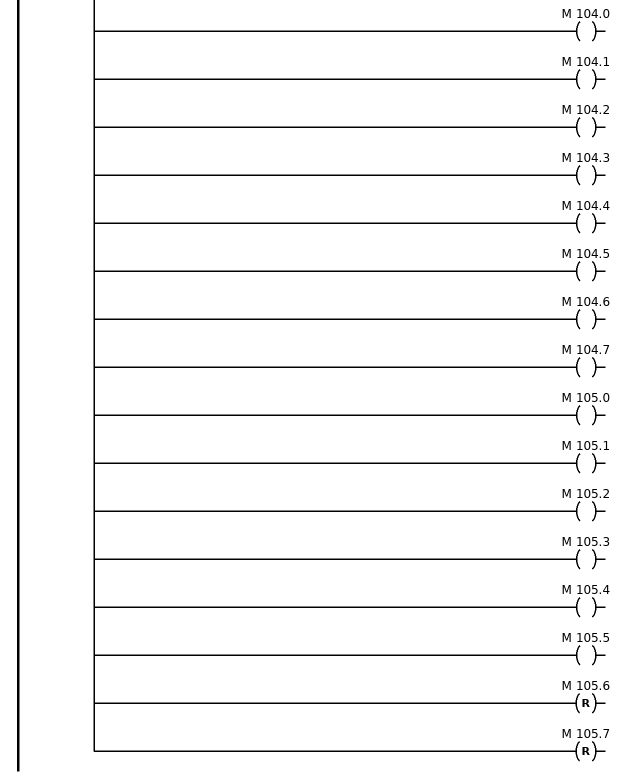
[picture p239: FC51 - TYPE TOOL networks 18-18]
NETWORK
TITLE = Error visible
      A     M 90.2;
      JCN   v10;
      SET;
      =     M 104.0;
      =     M 104.1;
      =     M 104.2;
      =     M 104.3;
      =     M 104.4;
      =     M 104.5;
      =     M 104.6;
      =     M 104.7;
      =     M 105.0;
      R     M 105.1;
      R     M 105.2;
      R     M 105.3;
      R     M 105.4;
      R     M 105.5;
      =     M 105.6;
      R     M 105.7;
      JU    next;
v10:  NOP   0;
      A     M 90.0;
      JCN   v11;
      SET;
      =     M 104.0;
      =     M 104.1;
      =     M 104.2;
      =     M 104.3;
      =     M 104.4;
      =     M 104.5;
      =     M 104.6;
      =     M 104.7;
      =     M 105.0;
      =     M 105.1;
      R     M 105.2;
      R     M 105.3;
      R     M 105.4;
      =     M 105.5;
      R     M 105.6;
      R     M 105.7;
      JU    next;
v11:  NOP   0;
      A     M 90.1;
      JCN   v13;
      SET;
      =     M 104.0;
      =     M 104.1;
      =     M 104.2;
      =     M 104.3;
      =     M 104.4;
      =     M 104.5;
      =     M 104.6;
      =     M 104.7;
      =     M 105.0;
      =     M 105.1;
      =     M 105.2;
      R     M 105.3;
      R     M 105.4;
      =     M 105.5;
      R     M 105.6;
      R     M 105.7;
      JU    next;
v13:  NOP   0;
      A     M 90.3;
      JCN   next;
      =     M 104.0;
      =     M 104.1;
      =     M 104.2;
      =     M 104.3;
      =     M 104.4;
      =     M 104.5;
      =     M 104.6;
      =     M 104.7;
      =     M 105.0;
      =     M 105.1;
      =     M 105.2;
      =     M 105.3;
      =     M 105.4;
      =     M 105.5;
      R     M 105.6;
      R     M 105.7;
next: NOP   0;
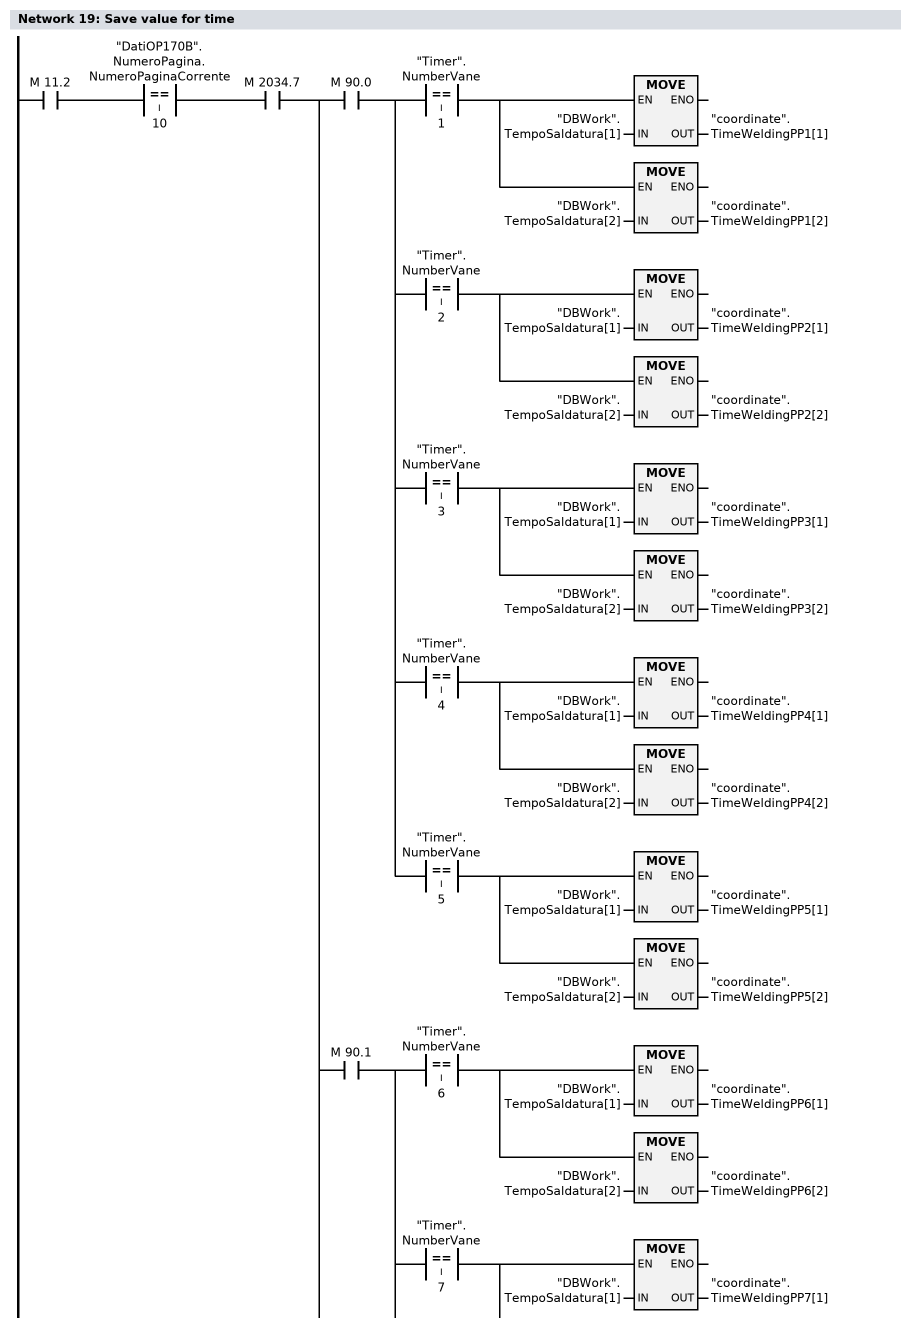
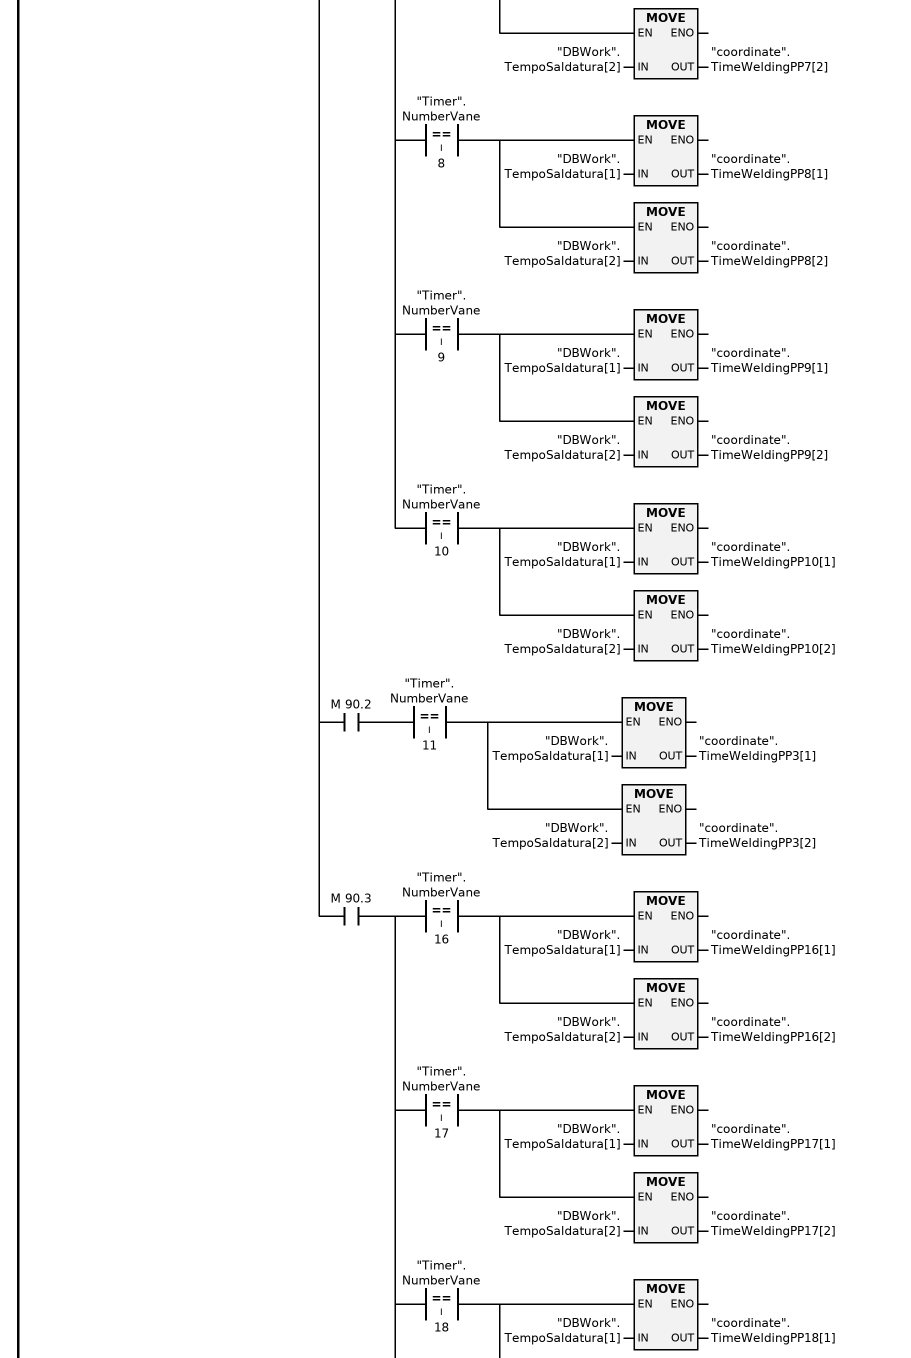
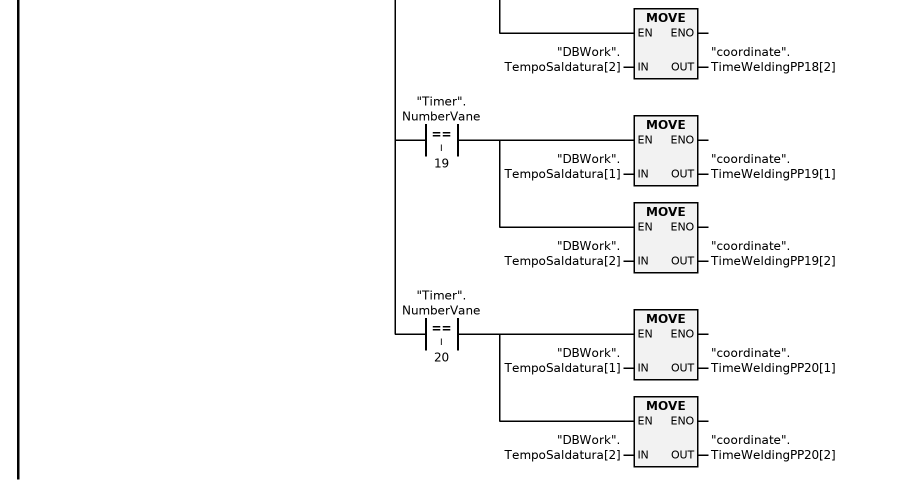
NETWORK
TITLE = Save value for time
      A     M 11.2;
      A(;
      L     "DatiOP170B".NumeroPagina.NumeroPaginaCorrente;
      L     10;
      ==I;
      );
      A     M 2034.7;
      =     L 0.0;
      A     L 0.0;
      A     M 90.0;
      =     L 0.1;
      A     L 0.1;
      A(;
      L     "Timer".NumberVane;
      L     1;
      ==I;
      );
      =     L 0.2;
      A     L 0.2;
      JNB   _0c6;
      L     "DBWork".TempoSaldatura[1];
      T     "coordinate".TimeWeldingPP1[1];
_0c6: NOP   0;
      A     L 0.2;
      JNB   _0c7;
      L     "DBWork".TempoSaldatura[2];
      T     "coordinate".TimeWeldingPP1[2];
_0c7: NOP   0;
      A     L 0.1;
      A(;
      L     "Timer".NumberVane;
      L     2;
      ==I;
      );
      =     L 0.2;
      A     L 0.2;
      JNB   _0c8;
      L     "DBWork".TempoSaldatura[1];
      T     "coordinate".TimeWeldingPP2[1];
_0c8: NOP   0;
      A     L 0.2;
      JNB   _0c9;
      L     "DBWork".TempoSaldatura[2];
      T     "coordinate".TimeWeldingPP2[2];
_0c9: NOP   0;
      A     L 0.1;
      A(;
      L     "Timer".NumberVane;
      L     3;
      ==I;
      );
      =     L 0.2;
      A     L 0.2;
      JNB   _0ca;
      L     "DBWork".TempoSaldatura[1];
      T     "coordinate".TimeWeldingPP3[1];
_0ca: NOP   0;
      A     L 0.2;
      JNB   _0cb;
      L     "DBWork".TempoSaldatura[2];
      T     "coordinate".TimeWeldingPP3[2];
_0cb: NOP   0;
      A     L 0.1;
      A(;
      L     "Timer".NumberVane;
      L     4;
      ==I;
      );
      =     L 0.2;
      A     L 0.2;
      JNB   _0cc;
      L     "DBWork".TempoSaldatura[1];
      T     "coordinate".TimeWeldingPP4[1];
_0cc: NOP   0;
      A     L 0.2;
      JNB   _0cd;
      L     "DBWork".TempoSaldatura[2];
      T     "coordinate".TimeWeldingPP4[2];
_0cd: NOP   0;
      A     L 0.1;
      A(;
      L     "Timer".NumberVane;
      L     5;
      ==I;
      );
      =     L 0.2;
      A     L 0.2;
      JNB   _0ce;
      L     "DBWork".TempoSaldatura[1];
      T     "coordinate".TimeWeldingPP5[1];
_0ce: NOP   0;
      A     L 0.2;
      JNB   _0cf;
      L     "DBWork".TempoSaldatura[2];
      T     "coordinate".TimeWeldingPP5[2];
_0cf: NOP   0;
      A     L 0.0;
      A     M 90.1;
      =     L 0.1;
      A     L 0.1;
      A(;
      L     "Timer".NumberVane;
      L     6;
      ==I;
      );
      =     L 0.2;
      A     L 0.2;
      JNB   _0d0;
      L     "DBWork".TempoSaldatura[1];
      T     "coordinate".TimeWeldingPP6[1];
_0d0: NOP   0;
      A     L 0.2;
      JNB   _0d1;
      L     "DBWork".TempoSaldatura[2];
      T     "coordinate".TimeWeldingPP6[2];
_0d1: NOP   0;
      A     L 0.1;
      A(;
      L     "Timer".NumberVane;
      L     7;
      ==I;
      );
      =     L 0.2;
      A     L 0.2;
      JNB   _0d2;
      L     "DBWork".TempoSaldatura[1];
      T     "coordinate".TimeWeldingPP7[1];
_0d2: NOP   0;
      A     L 0.2;
      JNB   _0d3;
      L     "DBWork".TempoSaldatura[2];
      T     "coordinate".TimeWeldingPP7[2];
_0d3: NOP   0;
      A     L 0.1;
      A(;
      L     "Timer".NumberVane;
      L     8;
      ==I;
      );
      =     L 0.2;
      A     L 0.2;
      JNB   _0d4;
      L     "DBWork".TempoSaldatura[1];
      T     "coordinate".TimeWeldingPP8[1];
_0d4: NOP   0;
      A     L 0.2;
      JNB   _0d5;
      L     "DBWork".TempoSaldatura[2];
      T     "coordinate".TimeWeldingPP8[2];
_0d5: NOP   0;
      A     L 0.1;
      A(;
      L     "Timer".NumberVane;
      L     9;
      ==I;
      );
      =     L 0.2;
      A     L 0.2;
      JNB   _0d6;
      L     "DBWork".TempoSaldatura[1];
      T     "coordinate".TimeWeldingPP9[1];
_0d6: NOP   0;
      A     L 0.2;
      JNB   _0d7;
      L     "DBWork".TempoSaldatura[2];
      T     "coordinate".TimeWeldingPP9[2];
_0d7: NOP   0;
      A     L 0.1;
      A(;
      L     "Timer".NumberVane;
      L     10;
      ==I;
      );
      =     L 0.2;
      A     L 0.2;
      JNB   _0d8;
      L     "DBWork".TempoSaldatura[1];
      T     "coordinate".TimeWeldingPP10[1];
_0d8: NOP   0;
      A     L 0.2;
      JNB   _0d9;
      L     "DBWork".TempoSaldatura[2];
      T     "coordinate".TimeWeldingPP10[2];
_0d9: NOP   0;
      A     L 0.0;
      A     M 90.2;
      A(;
      L     "Timer".NumberVane;
      L     11;
      ==I;
      );
      =     L 0.1;
      A     L 0.1;
      JNB   _0da;
      L     "DBWork".TempoSaldatura[1];
      T     "coordinate".TimeWeldingPP3[1];
_0da: NOP   0;
      A     L 0.1;
      JNB   _0db;
      L     "DBWork".TempoSaldatura[2];
      T     "coordinate".TimeWeldingPP3[2];
_0db: NOP   0;
      A     L 0.0;
      A     M 90.3;
      =     L 0.1;
      A     L 0.1;
      A(;
      L     "Timer".NumberVane;
      L     16;
      ==I;
      );
      =     L 0.2;
      A     L 0.2;
      JNB   _0dc;
      L     "DBWork".TempoSaldatura[1];
      T     "coordinate".TimeWeldingPP16[1];
_0dc: NOP   0;
      A     L 0.2;
      JNB   _0dd;
      L     "DBWork".TempoSaldatura[2];
      T     "coordinate".TimeWeldingPP16[2];
_0dd: NOP   0;
      A     L 0.1;
      A(;
      L     "Timer".NumberVane;
      L     17;
      ==I;
      );
      =     L 0.2;
      A     L 0.2;
      JNB   _0de;
      L     "DBWork".TempoSaldatura[1];
      T     "coordinate".TimeWeldingPP17[1];
_0de: NOP   0;
      A     L 0.2;
      JNB   _0df;
      L     "DBWork".TempoSaldatura[2];
      T     "coordinate".TimeWeldingPP17[2];
_0df: NOP   0;
      A     L 0.1;
      A(;
      L     "Timer".NumberVane;
      L     18;
      ==I;
      );
      =     L 0.2;
      A     L 0.2;
      JNB   _0e0;
      L     "DBWork".TempoSaldatura[1];
      T     "coordinate".TimeWeldingPP18[1];
_0e0: NOP   0;
      A     L 0.2;
      JNB   _0e1;
      L     "DBWork".TempoSaldatura[2];
      T     "coordinate".TimeWeldingPP18[2];
_0e1: NOP   0;
      A     L 0.1;
      A(;
      L     "Timer".NumberVane;
      L     19;
      ==I;
      );
      =     L 0.2;
      A     L 0.2;
      JNB   _0e2;
      L     "DBWork".TempoSaldatura[1];
      T     "coordinate".TimeWeldingPP19[1];
_0e2: NOP   0;
      A     L 0.2;
      JNB   _0e3;
      L     "DBWork".TempoSaldatura[2];
      T     "coordinate".TimeWeldingPP19[2];
_0e3: NOP   0;
      A     L 0.1;
      A(;
      L     "Timer".NumberVane;
      L     20;
      ==I;
      );
      =     L 0.2;
      A     L 0.2;
      JNB   _0e4;
      L     "DBWork".TempoSaldatura[1];
      T     "coordinate".TimeWeldingPP20[1];
_0e4: NOP   0;
      A     L 0.2;
      JNB   _0e5;
      L     "DBWork".TempoSaldatura[2];
      T     "coordinate".TimeWeldingPP20[2];
_0e5: NOP   0;
NETWORK
TITLE =
NETWORK
TITLE = load value for selected point, use it in auto, teach in and weld
//carico le coordinate del punto selezionato per fare le saldature in automatico 
//per il teachIn e per il test di salsatura
      A     M 1.1;
      =     L 0.0;
      A     L 0.0;
      A(;
      A(;
      L     "DBWork".PP[1].NumSaldaturaAtt;
      L     0;
      ==I;
      );
      A     M 11.4;
      O;
      A     M 11.2;
      A(;
      L     "DatiOP170B".PointWeldingTeachIn;
      L     1;
      ==I;
      );
      A(;
      O(;
      L     "DatiOP170B".NumeroPagina.NumeroPaginaCorrente;
      L     5;
      ==I;
      );
      O(;
      L     "DatiOP170B".NumeroPagina.NumeroPaginaCorrente;
      L     11;
      ==I;
      );
      );
      );
      =     L 0.1;
      A(;
      A     L 0.1;
      A     "DBWork".RotationTable;
      JNB   _0e6;
      L     "DBWork".CoordSaldatura[1].X1;
      T     MD 588;
      SET;
      SAVE;
      CLR;
_0e6: A     BR;
      );
      JNB   _0e7;
      L     "DBWork".CoordSaldatura[1].Y1;
      T     MD 592;
_0e7: NOP   0;
      A(;
      A     L 0.1;
      AN    "DBWork".RotationTable;
      JNB   _0e8;
      L     "DBWork".CoordSaldatura[1].X2;
      T     MD 588;
      SET;
      SAVE;
      CLR;
_0e8: A     BR;
      );
      JNB   _0e9;
      L     "DBWork".CoordSaldatura[1].Y2;
      T     MD 592;
_0e9: NOP   0;
      A     L 0.0;
      A(;
      A(;
      L     "DBWork".PP[1].NumSaldaturaAtt;
      L     1;
      ==I;
      );
      A     M 11.4;
      O;
      A     M 11.2;
      A(;
      L     "DatiOP170B".PointWeldingTeachIn;
      L     2;
      ==I;
      );
      A(;
      O(;
      L     "DatiOP170B".NumeroPagina.NumeroPaginaCorrente;
      L     5;
      ==I;
      );
      O(;
      L     "DatiOP170B".NumeroPagina.NumeroPaginaCorrente;
      L     11;
      ==I;
      );
      );
      );
      =     L 0.1;
      A(;
      A     L 0.1;
      A     "DBWork".RotationTable;
      JNB   _0ea;
      L     "DBWork".CoordSaldatura[2].X1;
      T     MD 588;
      SET;
      SAVE;
      CLR;
_0ea: A     BR;
      );
      JNB   _0eb;
      L     "DBWork".CoordSaldatura[2].Y1;
      T     MD 592;
_0eb: NOP   0;
      A(;
      A     L 0.1;
      AN    "DBWork".RotationTable;
      JNB   _0ec;
      L     "DBWork".CoordSaldatura[2].X2;
      T     MD 588;
      SET;
      SAVE;
      CLR;
_0ec: A     BR;
      );
      JNB   _0ed;
      L     "DBWork".CoordSaldatura[2].Y2;
      T     MD 592;
_0ed: NOP   0;
      A     L 0.0;
      A(;
      A(;
      L     "DBWork".PP[1].NumSaldaturaAtt;
      L     2;
      ==I;
      );
      A     M 11.4;
      O;
      A     M 11.2;
      A(;
      L     "DatiOP170B".PointWeldingTeachIn;
      L     3;
      ==I;
      );
      A(;
      O(;
      L     "DatiOP170B".NumeroPagina.NumeroPaginaCorrente;
      L     5;
      ==I;
      );
      O(;
      L     "DatiOP170B".NumeroPagina.NumeroPaginaCorrente;
      L     11;
      ==I;
      );
      );
      );
      =     L 0.1;
      A(;
      A     L 0.1;
      A     "DBWork".RotationTable;
      JNB   _0ee;
      L     "DBWork".CoordSaldatura[3].X1;
      T     MD 588;
      SET;
      SAVE;
      CLR;
_0ee: A     BR;
      );
      JNB   _0ef;
      L     "DBWork".CoordSaldatura[3].Y1;
      T     MD 592;
_0ef: NOP   0;
      A(;
      A     L 0.1;
      AN    "DBWork".RotationTable;
      JNB   _0f0;
      L     "DBWork".CoordSaldatura[3].X2;
      T     MD 588;
      SET;
      SAVE;
      CLR;
_0f0: A     BR;
      );
      JNB   _0f1;
      L     "DBWork".CoordSaldatura[3].Y2;
      T     MD 592;
_0f1: NOP   0;
      A     L 0.0;
      A(;
      A(;
      L     "DBWork".PP[1].NumSaldaturaAtt;
      L     3;
      ==I;
      );
      A     M 11.4;
      O;
      A     M 11.2;
      A(;
      L     "DatiOP170B".PointWeldingTeachIn;
      L     4;
      ==I;
      );
      A(;
      O(;
      L     "DatiOP170B".NumeroPagina.NumeroPaginaCorrente;
      L     5;
      ==I;
      );
      O(;
      L     "DatiOP170B".NumeroPagina.NumeroPaginaCorrente;
      L     11;
      ==I;
      );
      );
      );
      =     L 0.1;
      A(;
      A     L 0.1;
      A     "DBWork".RotationTable;
      JNB   _0f2;
      L     "DBWork".CoordSaldatura[4].X1;
      T     MD 588;
      SET;
      SAVE;
      CLR;
_0f2: A     BR;
      );
      JNB   _0f3;
      L     "DBWork".CoordSaldatura[4].Y1;
      T     MD 592;
_0f3: NOP   0;
      A(;
      A     L 0.1;
      AN    "DBWork".RotationTable;
      JNB   _0f4;
      L     "DBWork".CoordSaldatura[4].X2;
      T     MD 588;
      SET;
      SAVE;
      CLR;
_0f4: A     BR;
      );
      JNB   _0f5;
      L     "DBWork".CoordSaldatura[4].Y2;
      T     MD 592;
_0f5: NOP   0;
      A     L 0.0;
      A(;
      A(;
      L     "DBWork".PP[1].NumSaldaturaAtt;
      L     4;
      ==I;
      );
      A     M 11.4;
      O;
      A     M 11.2;
      A(;
      L     "DatiOP170B".PointWeldingTeachIn;
      L     5;
      ==I;
      );
      A(;
      O(;
      L     "DatiOP170B".NumeroPagina.NumeroPaginaCorrente;
      L     5;
      ==I;
      );
      O(;
      L     "DatiOP170B".NumeroPagina.NumeroPaginaCorrente;
      L     11;
      ==I;
      );
      );
      );
      =     L 0.1;
      A(;
      A     L 0.1;
      A     "DBWork".RotationTable;
      JNB   _0f6;
      L     "DBWork".CoordSaldatura[5].X1;
      T     MD 588;
      SET;
      SAVE;
      CLR;
_0f6: A     BR;
      );
      JNB   _0f7;
      L     "DBWork".CoordSaldatura[5].Y1;
      T     MD 592;
_0f7: NOP   0;
      A(;
      A     L 0.1;
      AN    "DBWork".RotationTable;
      JNB   _0f8;
      L     "DBWork".CoordSaldatura[5].X2;
      T     MD 588;
      SET;
      SAVE;
      CLR;
_0f8: A     BR;
      );
      JNB   _0f9;
      L     "DBWork".CoordSaldatura[5].Y2;
      T     MD 592;
_0f9: NOP   0;
      A     L 0.0;
      A(;
      A(;
      L     "DBWork".PP[1].NumSaldaturaAtt;
      L     5;
      ==I;
      );
      A     M 11.4;
      O;
      A     M 11.2;
      A(;
      L     "DatiOP170B".PointWeldingTeachIn;
      L     6;
      ==I;
      );
      A(;
      O(;
      L     "DatiOP170B".NumeroPagina.NumeroPaginaCorrente;
      L     5;
      ==I;
      );
      O(;
      L     "DatiOP170B".NumeroPagina.NumeroPaginaCorrente;
      L     11;
      ==I;
      );
      );
      );
      =     L 0.1;
      A(;
      A     L 0.1;
      A     "DBWork".RotationTable;
      JNB   _0fa;
      L     "DBWork".CoordSaldatura[6].X1;
      T     MD 588;
      SET;
      SAVE;
      CLR;
_0fa: A     BR;
      );
      JNB   _0fb;
      L     "DBWork".CoordSaldatura[6].Y1;
      T     MD 592;
_0fb: NOP   0;
      A(;
      A     L 0.1;
      AN    "DBWork".RotationTable;
      JNB   _0fc;
      L     "DBWork".CoordSaldatura[6].X2;
      T     MD 588;
      SET;
      SAVE;
      CLR;
_0fc: A     BR;
      );
      JNB   _0fd;
      L     "DBWork".CoordSaldatura[6].Y2;
      T     MD 592;
_0fd: NOP   0;
      A     L 0.0;
      A(;
      A(;
      L     "DBWork".PP[1].NumSaldaturaAtt;
      L     6;
      ==I;
      );
      A     M 11.4;
      O;
      A     M 11.2;
      A(;
      L     "DatiOP170B".PointWeldingTeachIn;
      L     7;
      ==I;
      );
      A(;
      O(;
      L     "DatiOP170B".NumeroPagina.NumeroPaginaCorrente;
      L     5;
      ==I;
      );
      O(;
      L     "DatiOP170B".NumeroPagina.NumeroPaginaCorrente;
      L     11;
      ==I;
      );
      );
      );
      =     L 0.1;
      A(;
      A     L 0.1;
      A     "DBWork".RotationTable;
      JNB   _0fe;
      L     "DBWork".CoordSaldatura[7].X1;
      T     MD 588;
      SET;
      SAVE;
      CLR;
_0fe: A     BR;
      );
      JNB   _0ff;
      L     "DBWork".CoordSaldatura[7].Y1;
      T     MD 592;
_0ff: NOP   0;
      A(;
      A     L 0.1;
      AN    "DBWork".RotationTable;
      JNB   _100;
      L     "DBWork".CoordSaldatura[7].X2;
      T     MD 588;
      SET;
      SAVE;
      CLR;
_100: A     BR;
      );
      JNB   _101;
      L     "DBWork".CoordSaldatura[7].Y2;
      T     MD 592;
_101: NOP   0;
      A     L 0.0;
      A(;
      A(;
      L     "DBWork".PP[1].NumSaldaturaAtt;
      L     7;
      ==I;
      );
      A     M 11.4;
      O;
      A     M 11.2;
      A(;
      L     "DatiOP170B".PointWeldingTeachIn;
      L     8;
      ==I;
      );
      A(;
      O(;
      L     "DatiOP170B".NumeroPagina.NumeroPaginaCorrente;
      L     5;
      ==I;
      );
      O(;
      L     "DatiOP170B".NumeroPagina.NumeroPaginaCorrente;
      L     11;
      ==I;
      );
      );
      );
      =     L 0.1;
      A(;
      A     L 0.1;
      A     "DBWork".RotationTable;
      JNB   _102;
      L     "DBWork".CoordSaldatura[8].X1;
      T     MD 588;
      SET;
      SAVE;
      CLR;
_102: A     BR;
      );
      JNB   _103;
      L     "DBWork".CoordSaldatura[8].Y1;
      T     MD 592;
_103: NOP   0;
      A(;
      A     L 0.1;
      AN    "DBWork".RotationTable;
      JNB   _104;
      L     "DBWork".CoordSaldatura[8].X2;
      T     MD 588;
      SET;
      SAVE;
      CLR;
_104: A     BR;
      );
      JNB   _105;
      L     "DBWork".CoordSaldatura[8].Y2;
      T     MD 592;
_105: NOP   0;
      A     L 0.0;
      A(;
      A(;
      L     "DBWork".PP[1].NumSaldaturaAtt;
      L     8;
      ==I;
      );
      A     M 11.4;
      O;
      A     M 11.2;
      A(;
      L     "DatiOP170B".PointWeldingTeachIn;
      L     9;
      ==I;
      );
      A(;
      O(;
      L     "DatiOP170B".NumeroPagina.NumeroPaginaCorrente;
      L     5;
      ==I;
      );
      O(;
      L     "DatiOP170B".NumeroPagina.NumeroPaginaCorrente;
      L     11;
      ==I;
      );
      );
      );
      =     L 0.1;
      A(;
      A     L 0.1;
      A     "DBWork".RotationTable;
      JNB   _106;
      L     "DBWork".CoordSaldatura[9].X1;
      T     MD 588;
      SET;
      SAVE;
      CLR;
_106: A     BR;
      );
      JNB   _107;
      L     "DBWork".CoordSaldatura[9].Y1;
      T     MD 592;
_107: NOP   0;
      A(;
      A     L 0.1;
      AN    "DBWork".RotationTable;
      JNB   _108;
      L     "DBWork".CoordSaldatura[9].X2;
      T     MD 588;
      SET;
      SAVE;
      CLR;
_108: A     BR;
      );
      JNB   _109;
      L     "DBWork".CoordSaldatura[9].Y2;
      T     MD 592;
_109: NOP   0;
      A     L 0.0;
      A(;
      A(;
      L     "DBWork".PP[1].NumSaldaturaAtt;
      L     9;
      ==I;
      );
      A     M 11.4;
      O;
      A     M 11.2;
      A(;
      L     "DatiOP170B".PointWeldingTeachIn;
      L     10;
      ==I;
      );
      A(;
      O(;
      L     "DatiOP170B".NumeroPagina.NumeroPaginaCorrente;
      L     5;
      ==I;
      );
      O(;
      L     "DatiOP170B".NumeroPagina.NumeroPaginaCorrente;
      L     11;
      ==I;
      );
      );
      );
      =     L 0.1;
      A(;
      A     L 0.1;
      A     "DBWork".RotationTable;
      JNB   _10a;
      L     "DBWork".CoordSaldatura[10].X1;
      T     MD 588;
      SET;
      SAVE;
      CLR;
_10a: A     BR;
      );
      JNB   _10b;
      L     "DBWork".CoordSaldatura[10].Y1;
      T     MD 592;
_10b: NOP   0;
      A(;
      A     L 0.1;
      AN    "DBWork".RotationTable;
      JNB   _10c;
      L     "DBWork".CoordSaldatura[10].X2;
      T     MD 588;
      SET;
      SAVE;
      CLR;
_10c: A     BR;
      );
      JNB   _10d;
      L     "DBWork".CoordSaldatura[10].Y2;
      T     MD 592;
_10d: NOP   0;
      A     L 0.0;
      A(;
      A(;
      L     "DBWork".PP[1].NumSaldaturaAtt;
      L     10;
      ==I;
      );
      A     M 11.4;
      O;
      A     M 11.2;
      A(;
      L     "DatiOP170B".PointWeldingTeachIn;
      L     11;
      ==I;
      );
      A(;
      O(;
      L     "DatiOP170B".NumeroPagina.NumeroPaginaCorrente;
      L     5;
      ==I;
      );
      O(;
      L     "DatiOP170B".NumeroPagina.NumeroPaginaCorrente;
      L     11;
      ==I;
      );
      );
      );
      =     L 0.1;
      A(;
      A     L 0.1;
      A     "DBWork".RotationTable;
      JNB   _10e;
      L     "DBWork".CoordSaldatura[11].X1;
      T     MD 588;
      SET;
      SAVE;
      CLR;
_10e: A     BR;
      );
      JNB   _10f;
      L     "DBWork".CoordSaldatura[11].Y1;
      T     MD 592;
_10f: NOP   0;
      A(;
      A     L 0.1;
      AN    "DBWork".RotationTable;
      JNB   _110;
      L     "DBWork".CoordSaldatura[11].X2;
      T     MD 588;
      SET;
      SAVE;
      CLR;
_110: A     BR;
      );
      JNB   _111;
      L     "DBWork".CoordSaldatura[11].Y2;
      T     MD 592;
_111: NOP   0;
      A     L 0.0;
      A(;
      A(;
      L     "DBWork".PP[1].NumSaldaturaAtt;
      L     11;
      ==I;
      );
      A     M 11.4;
      O;
      A     M 11.2;
      A(;
      L     "DatiOP170B".PointWeldingTeachIn;
      L     12;
      ==I;
      );
      A(;
      O(;
      L     "DatiOP170B".NumeroPagina.NumeroPaginaCorrente;
      L     5;
      ==I;
      );
      O(;
      L     "DatiOP170B".NumeroPagina.NumeroPaginaCorrente;
      L     11;
      ==I;
      );
      );
      );
      =     L 0.1;
      A(;
      A     L 0.1;
      A     "DBWork".RotationTable;
      JNB   _112;
      L     "DBWork".CoordSaldatura[12].X1;
      T     MD 588;
      SET;
      SAVE;
      CLR;
_112: A     BR;
      );
      JNB   _113;
      L     "DBWork".CoordSaldatura[12].Y1;
      T     MD 592;
_113: NOP   0;
      A(;
      A     L 0.1;
      AN    "DBWork".RotationTable;
      JNB   _114;
      L     "DBWork".CoordSaldatura[12].X2;
      T     MD 588;
      SET;
      SAVE;
      CLR;
_114: A     BR;
      );
      JNB   _115;
      L     "DBWork".CoordSaldatura[12].Y2;
      T     MD 592;
_115: NOP   0;
      A     L 0.0;
      A(;
      A(;
      L     "DBWork".PP[1].NumSaldaturaAtt;
      L     12;
      ==I;
      );
      A     M 11.4;
      O;
      A     M 11.2;
      A(;
      L     "DatiOP170B".PointWeldingTeachIn;
      L     13;
      ==I;
      );
      A(;
      O(;
      L     "DatiOP170B".NumeroPagina.NumeroPaginaCorrente;
      L     5;
      ==I;
      );
      O(;
      L     "DatiOP170B".NumeroPagina.NumeroPaginaCorrente;
      L     11;
      ==I;
      );
      );
      );
      =     L 0.1;
      A(;
      A     L 0.1;
      A     "DBWork".RotationTable;
      JNB   _116;
      L     "DBWork".CoordSaldatura[13].X1;
      T     MD 588;
      SET;
      SAVE;
      CLR;
_116: A     BR;
      );
      JNB   _117;
      L     "DBWork".CoordSaldatura[13].Y1;
      T     MD 592;
_117: NOP   0;
      A(;
      A     L 0.1;
      AN    "DBWork".RotationTable;
      JNB   _118;
      L     "DBWork".CoordSaldatura[13].X2;
      T     MD 588;
      SET;
      SAVE;
      CLR;
_118: A     BR;
      );
      JNB   _119;
      L     "DBWork".CoordSaldatura[13].Y2;
      T     MD 592;
_119: NOP   0;
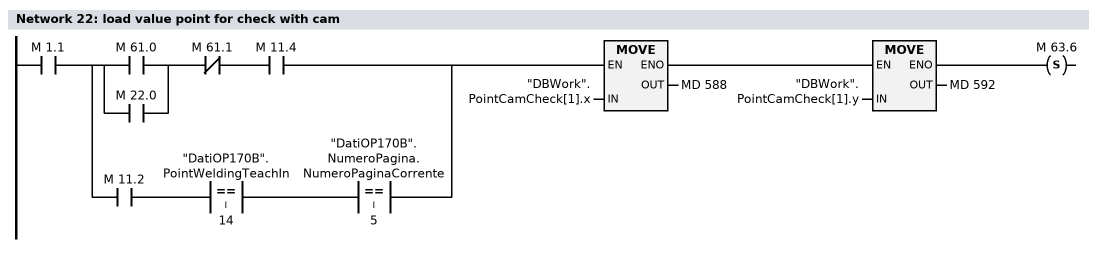
NETWORK
TITLE = load value point for check with cam
//posizione per fare la foto
      A(;
      A     M 1.1;
      A(;
      A(;
      O     M 61.0;
      O     M 22.0;
      );
      AN    M 61.1;
      A     M 11.4;
      O;
      A     M 11.2;
      A(;
      L     "DatiOP170B".PointWeldingTeachIn;
      L     14;
      ==I;
      );
      A(;
      L     "DatiOP170B".NumeroPagina.NumeroPaginaCorrente;
      L     5;
      ==I;
      );
      );
      JNB   _11a;
      L     "DBWork".PointCamCheck[1].x;
      T     MD 588;
      SET;
      SAVE;
      CLR;
_11a: A     BR;
      );
      JNB   _11b;
      L     "DBWork".PointCamCheck[1].y;
      T     MD 592;
      SET;
      SAVE;
      CLR;
_11b: A     BR;
      S     M 63.6;
NETWORK
TITLE = ******************** Value point for Welding *******A***********
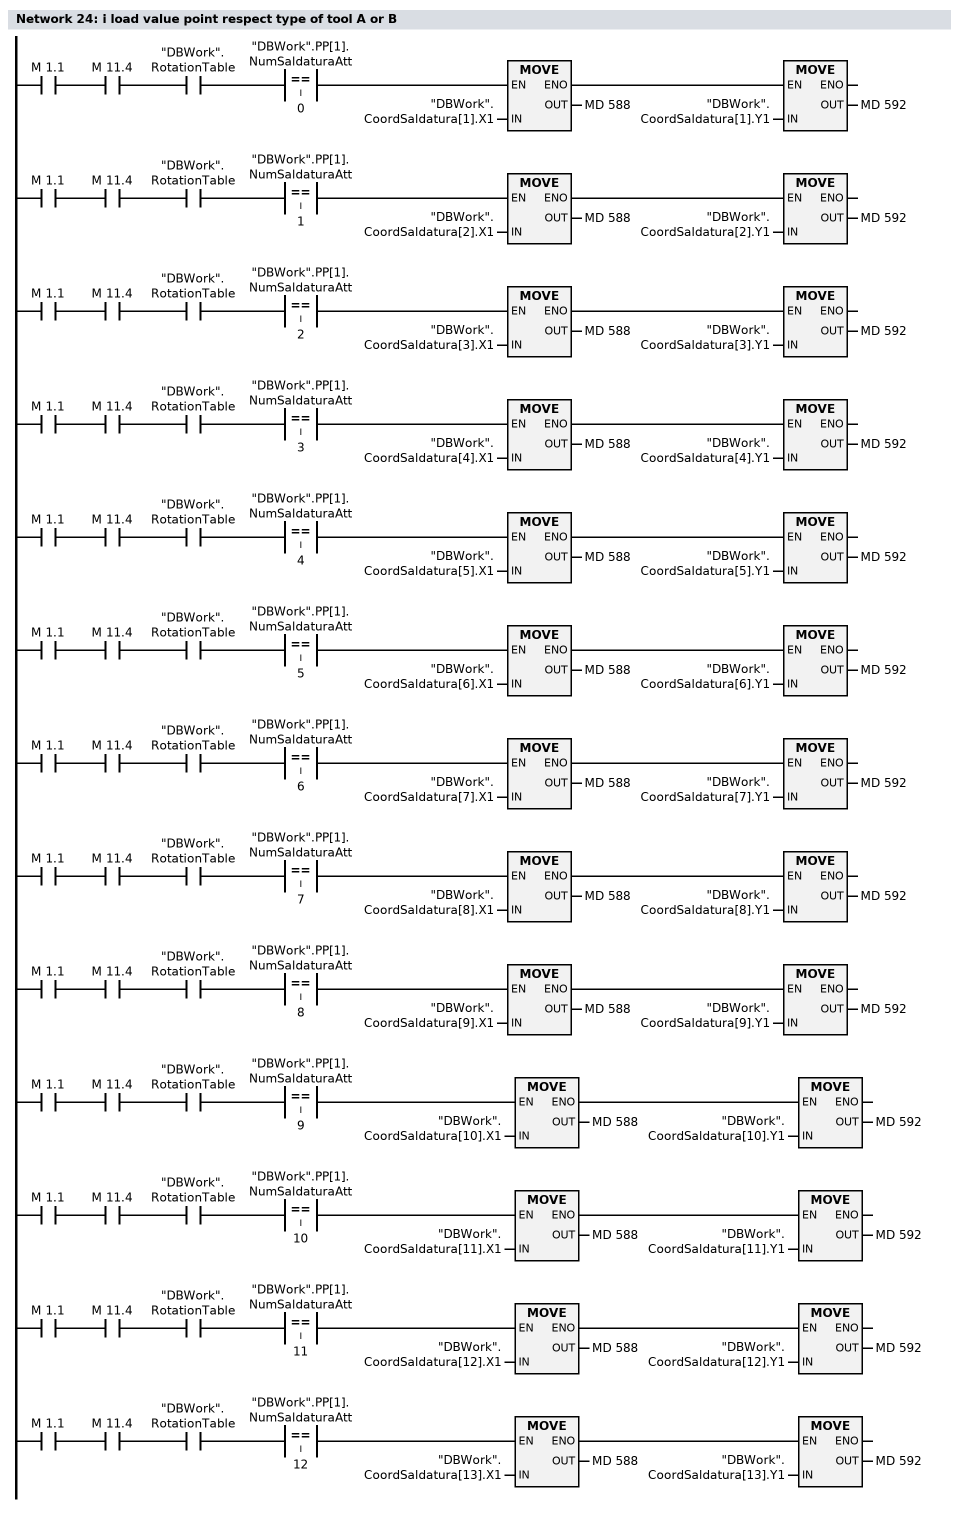
NETWORK
TITLE = i load value point respect type of tool A or B
//In base alla saldatura che effettuo passo le coordinate a gli assi
      A     M 1.1;
      A     M 11.4;
      A     "DBWork".RotationTable;
      =     L 0.0;
      A(;
      A     L 0.0;
      A(;
      L     "DBWork".PP[1].NumSaldaturaAtt;
      L     0;
      ==I;
      );
      JNB   _11c;
      L     "DBWork".CoordSaldatura[1].X1;
      T     MD 588;
      SET;
      SAVE;
      CLR;
_11c: A     BR;
      );
      JNB   _11d;
      L     "DBWork".CoordSaldatura[1].Y1;
      T     MD 592;
_11d: NOP   0;
      A(;
      A     L 0.0;
      A(;
      L     "DBWork".PP[1].NumSaldaturaAtt;
      L     1;
      ==I;
      );
      JNB   _11e;
      L     "DBWork".CoordSaldatura[2].X1;
      T     MD 588;
      SET;
      SAVE;
      CLR;
_11e: A     BR;
      );
      JNB   _11f;
      L     "DBWork".CoordSaldatura[2].Y1;
      T     MD 592;
_11f: NOP   0;
      A(;
      A     L 0.0;
      A(;
      L     "DBWork".PP[1].NumSaldaturaAtt;
      L     2;
      ==I;
      );
      JNB   _120;
      L     "DBWork".CoordSaldatura[3].X1;
      T     MD 588;
      SET;
      SAVE;
      CLR;
_120: A     BR;
      );
      JNB   _121;
      L     "DBWork".CoordSaldatura[3].Y1;
      T     MD 592;
_121: NOP   0;
      A(;
      A     L 0.0;
      A(;
      L     "DBWork".PP[1].NumSaldaturaAtt;
      L     3;
      ==I;
      );
      JNB   _122;
      L     "DBWork".CoordSaldatura[4].X1;
      T     MD 588;
      SET;
      SAVE;
      CLR;
_122: A     BR;
      );
      JNB   _123;
      L     "DBWork".CoordSaldatura[4].Y1;
      T     MD 592;
_123: NOP   0;
      A(;
      A     L 0.0;
      A(;
      L     "DBWork".PP[1].NumSaldaturaAtt;
      L     4;
      ==I;
      );
      JNB   _124;
      L     "DBWork".CoordSaldatura[5].X1;
      T     MD 588;
      SET;
      SAVE;
      CLR;
_124: A     BR;
      );
      JNB   _125;
      L     "DBWork".CoordSaldatura[5].Y1;
      T     MD 592;
_125: NOP   0;
      A(;
      A     L 0.0;
      A(;
      L     "DBWork".PP[1].NumSaldaturaAtt;
      L     5;
      ==I;
      );
      JNB   _126;
      L     "DBWork".CoordSaldatura[6].X1;
      T     MD 588;
      SET;
      SAVE;
      CLR;
_126: A     BR;
      );
      JNB   _127;
      L     "DBWork".CoordSaldatura[6].Y1;
      T     MD 592;
_127: NOP   0;
      A(;
      A     L 0.0;
      A(;
      L     "DBWork".PP[1].NumSaldaturaAtt;
      L     6;
      ==I;
      );
      JNB   _128;
      L     "DBWork".CoordSaldatura[7].X1;
      T     MD 588;
      SET;
      SAVE;
      CLR;
_128: A     BR;
      );
      JNB   _129;
      L     "DBWork".CoordSaldatura[7].Y1;
      T     MD 592;
_129: NOP   0;
      A(;
      A     L 0.0;
      A(;
      L     "DBWork".PP[1].NumSaldaturaAtt;
      L     7;
      ==I;
      );
      JNB   _12a;
      L     "DBWork".CoordSaldatura[8].X1;
      T     MD 588;
      SET;
      SAVE;
      CLR;
_12a: A     BR;
      );
      JNB   _12b;
      L     "DBWork".CoordSaldatura[8].Y1;
      T     MD 592;
_12b: NOP   0;
      A(;
      A     L 0.0;
      A(;
      L     "DBWork".PP[1].NumSaldaturaAtt;
      L     8;
      ==I;
      );
      JNB   _12c;
      L     "DBWork".CoordSaldatura[9].X1;
      T     MD 588;
      SET;
      SAVE;
      CLR;
_12c: A     BR;
      );
      JNB   _12d;
      L     "DBWork".CoordSaldatura[9].Y1;
      T     MD 592;
_12d: NOP   0;
      A(;
      A     L 0.0;
      A(;
      L     "DBWork".PP[1].NumSaldaturaAtt;
      L     9;
      ==I;
      );
      JNB   _12e;
      L     "DBWork".CoordSaldatura[10].X1;
      T     MD 588;
      SET;
      SAVE;
      CLR;
_12e: A     BR;
      );
      JNB   _12f;
      L     "DBWork".CoordSaldatura[10].Y1;
      T     MD 592;
_12f: NOP   0;
      A(;
      A     L 0.0;
      A(;
      L     "DBWork".PP[1].NumSaldaturaAtt;
      L     10;
      ==I;
      );
      JNB   _130;
      L     "DBWork".CoordSaldatura[11].X1;
      T     MD 588;
      SET;
      SAVE;
      CLR;
_130: A     BR;
      );
      JNB   _131;
      L     "DBWork".CoordSaldatura[11].Y1;
      T     MD 592;
_131: NOP   0;
      A(;
      A     L 0.0;
      A(;
      L     "DBWork".PP[1].NumSaldaturaAtt;
      L     11;
      ==I;
      );
      JNB   _132;
      L     "DBWork".CoordSaldatura[12].X1;
      T     MD 588;
      SET;
      SAVE;
      CLR;
_132: A     BR;
      );
      JNB   _133;
      L     "DBWork".CoordSaldatura[12].Y1;
      T     MD 592;
_133: NOP   0;
      A(;
      A     L 0.0;
      A(;
      L     "DBWork".PP[1].NumSaldaturaAtt;
      L     12;
      ==I;
      );
      JNB   _134;
      L     "DBWork".CoordSaldatura[13].X1;
      T     MD 588;
      SET;
      SAVE;
      CLR;
_134: A     BR;
      );
      JNB   _135;
      L     "DBWork".CoordSaldatura[13].Y1;
      T     MD 592;
_135: NOP   0;
NETWORK
TITLE = ******************** Value Point for Welding *********B********
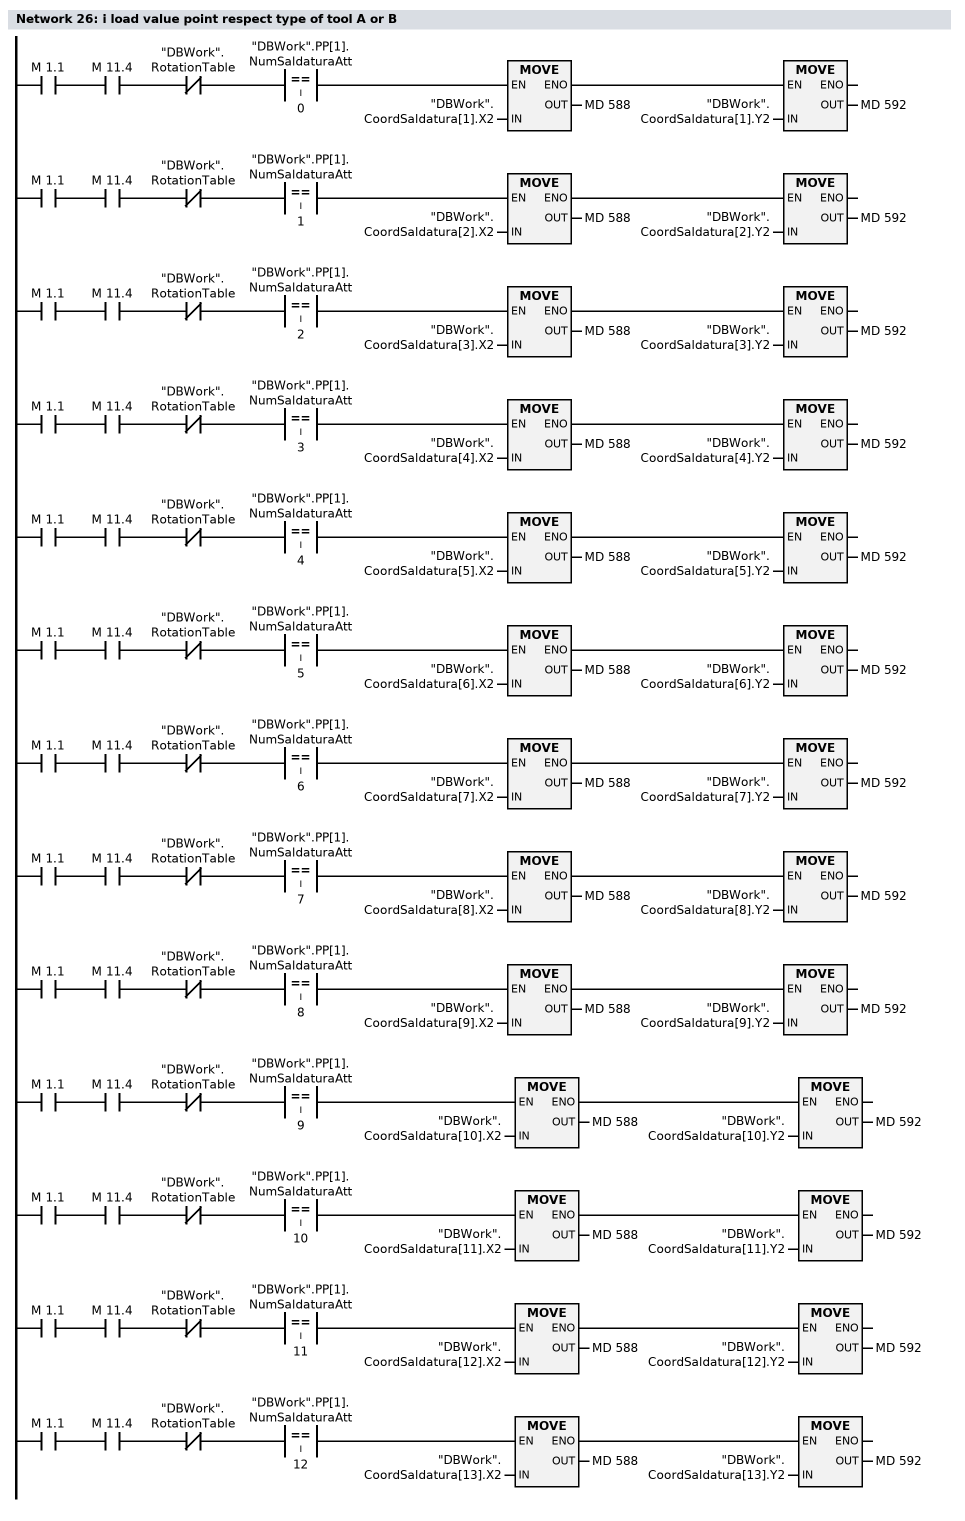
NETWORK
TITLE = i load value point respect type of tool A or B
//In base alla saldatura che effettuo passo le coordinate a gli assi
      A     M 1.1;
      A     M 11.4;
      AN    "DBWork".RotationTable;
      =     L 0.0;
      A(;
      A     L 0.0;
      A(;
      L     "DBWork".PP[1].NumSaldaturaAtt;
      L     0;
      ==I;
      );
      JNB   _136;
      L     "DBWork".CoordSaldatura[1].X2;
      T     MD 588;
      SET;
      SAVE;
      CLR;
_136: A     BR;
      );
      JNB   _137;
      L     "DBWork".CoordSaldatura[1].Y2;
      T     MD 592;
_137: NOP   0;
      A(;
      A     L 0.0;
      A(;
      L     "DBWork".PP[1].NumSaldaturaAtt;
      L     1;
      ==I;
      );
      JNB   _138;
      L     "DBWork".CoordSaldatura[2].X2;
      T     MD 588;
      SET;
      SAVE;
      CLR;
_138: A     BR;
      );
      JNB   _139;
      L     "DBWork".CoordSaldatura[2].Y2;
      T     MD 592;
_139: NOP   0;
      A(;
      A     L 0.0;
      A(;
      L     "DBWork".PP[1].NumSaldaturaAtt;
      L     2;
      ==I;
      );
      JNB   _13a;
      L     "DBWork".CoordSaldatura[3].X2;
      T     MD 588;
      SET;
      SAVE;
      CLR;
_13a: A     BR;
      );
      JNB   _13b;
      L     "DBWork".CoordSaldatura[3].Y2;
      T     MD 592;
_13b: NOP   0;
      A(;
      A     L 0.0;
      A(;
      L     "DBWork".PP[1].NumSaldaturaAtt;
      L     3;
      ==I;
      );
      JNB   _13c;
      L     "DBWork".CoordSaldatura[4].X2;
      T     MD 588;
      SET;
      SAVE;
      CLR;
_13c: A     BR;
      );
      JNB   _13d;
      L     "DBWork".CoordSaldatura[4].Y2;
      T     MD 592;
_13d: NOP   0;
      A(;
      A     L 0.0;
      A(;
      L     "DBWork".PP[1].NumSaldaturaAtt;
      L     4;
      ==I;
      );
      JNB   _13e;
      L     "DBWork".CoordSaldatura[5].X2;
      T     MD 588;
      SET;
      SAVE;
      CLR;
_13e: A     BR;
      );
      JNB   _13f;
      L     "DBWork".CoordSaldatura[5].Y2;
      T     MD 592;
_13f: NOP   0;
      A(;
      A     L 0.0;
      A(;
      L     "DBWork".PP[1].NumSaldaturaAtt;
      L     5;
      ==I;
      );
      JNB   _140;
      L     "DBWork".CoordSaldatura[6].X2;
      T     MD 588;
      SET;
      SAVE;
      CLR;
_140: A     BR;
      );
      JNB   _141;
      L     "DBWork".CoordSaldatura[6].Y2;
      T     MD 592;
_141: NOP   0;
      A(;
      A     L 0.0;
      A(;
      L     "DBWork".PP[1].NumSaldaturaAtt;
      L     6;
      ==I;
      );
      JNB   _142;
      L     "DBWork".CoordSaldatura[7].X2;
      T     MD 588;
      SET;
      SAVE;
      CLR;
_142: A     BR;
      );
      JNB   _143;
      L     "DBWork".CoordSaldatura[7].Y2;
      T     MD 592;
_143: NOP   0;
      A(;
      A     L 0.0;
      A(;
      L     "DBWork".PP[1].NumSaldaturaAtt;
      L     7;
      ==I;
      );
      JNB   _144;
      L     "DBWork".CoordSaldatura[8].X2;
      T     MD 588;
      SET;
      SAVE;
      CLR;
_144: A     BR;
      );
      JNB   _145;
      L     "DBWork".CoordSaldatura[8].Y2;
      T     MD 592;
_145: NOP   0;
      A(;
      A     L 0.0;
      A(;
      L     "DBWork".PP[1].NumSaldaturaAtt;
      L     8;
      ==I;
      );
      JNB   _146;
      L     "DBWork".CoordSaldatura[9].X2;
      T     MD 588;
      SET;
      SAVE;
      CLR;
_146: A     BR;
      );
      JNB   _147;
      L     "DBWork".CoordSaldatura[9].Y2;
      T     MD 592;
_147: NOP   0;
      A(;
      A     L 0.0;
      A(;
      L     "DBWork".PP[1].NumSaldaturaAtt;
      L     9;
      ==I;
      );
      JNB   _148;
      L     "DBWork".CoordSaldatura[10].X2;
      T     MD 588;
      SET;
      SAVE;
      CLR;
_148: A     BR;
      );
      JNB   _149;
      L     "DBWork".CoordSaldatura[10].Y2;
      T     MD 592;
_149: NOP   0;
      A(;
      A     L 0.0;
      A(;
      L     "DBWork".PP[1].NumSaldaturaAtt;
      L     10;
      ==I;
      );
      JNB   _14a;
      L     "DBWork".CoordSaldatura[11].X2;
      T     MD 588;
      SET;
      SAVE;
      CLR;
_14a: A     BR;
      );
      JNB   _14b;
      L     "DBWork".CoordSaldatura[11].Y2;
      T     MD 592;
_14b: NOP   0;
      A(;
      A     L 0.0;
      A(;
      L     "DBWork".PP[1].NumSaldaturaAtt;
      L     11;
      ==I;
      );
      JNB   _14c;
      L     "DBWork".CoordSaldatura[12].X2;
      T     MD 588;
      SET;
      SAVE;
      CLR;
_14c: A     BR;
      );
      JNB   _14d;
      L     "DBWork".CoordSaldatura[12].Y2;
      T     MD 592;
_14d: NOP   0;
      A(;
      A     L 0.0;
      A(;
      L     "DBWork".PP[1].NumSaldaturaAtt;
      L     12;
      ==I;
      );
      JNB   _14e;
      L     "DBWork".CoordSaldatura[13].X2;
      T     MD 588;
      SET;
      SAVE;
      CLR;
_14e: A     BR;
      );
      JNB   _14f;
      L     "DBWork".CoordSaldatura[13].Y2;
      T     MD 592;
_14f: NOP   0;
NETWORK
TITLE = ******************** Point for Vision **************************
END_FUNCTION

FUNCTION "FC52 - SYSTEM VISION" : VOID	// FC 52
VERSION : 0.1
BEGIN
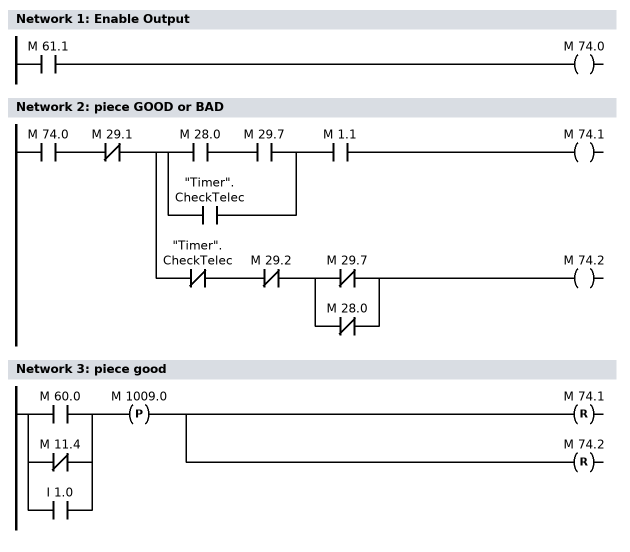
NETWORK
TITLE = Enable Output 
      A     M 61.1;
      =     M 74.0;
NETWORK
TITLE = piece GOOD or BAD
      A     M 74.0;
      AN    M 29.1;
      =     L 0.0;
      A     L 0.0;
      A(;
      A     M 28.0;
      A     M 29.7;
      O     "Timer".CheckTelec;
      );
      A     M 1.1;
      =     M 74.1;
      A     L 0.0;
      AN    "Timer".CheckTelec;
      AN    M 29.2;
      A(;
      ON    M 29.7;
      ON    M 28.0;
      );
      =     M 74.2;
NETWORK
TITLE = piece good
      A(;
      O     M 60.0;
      ON    M 11.4;
      O     I 1.0;
      );
      FP    M 1009.0;
      R     M 74.1;
      R     M 74.2;
END_FUNCTION

FUNCTION "FC53 - REWORK" : VOID	// FC 53
VERSION : 0.1
BEGIN
NETWORK
TITLE =
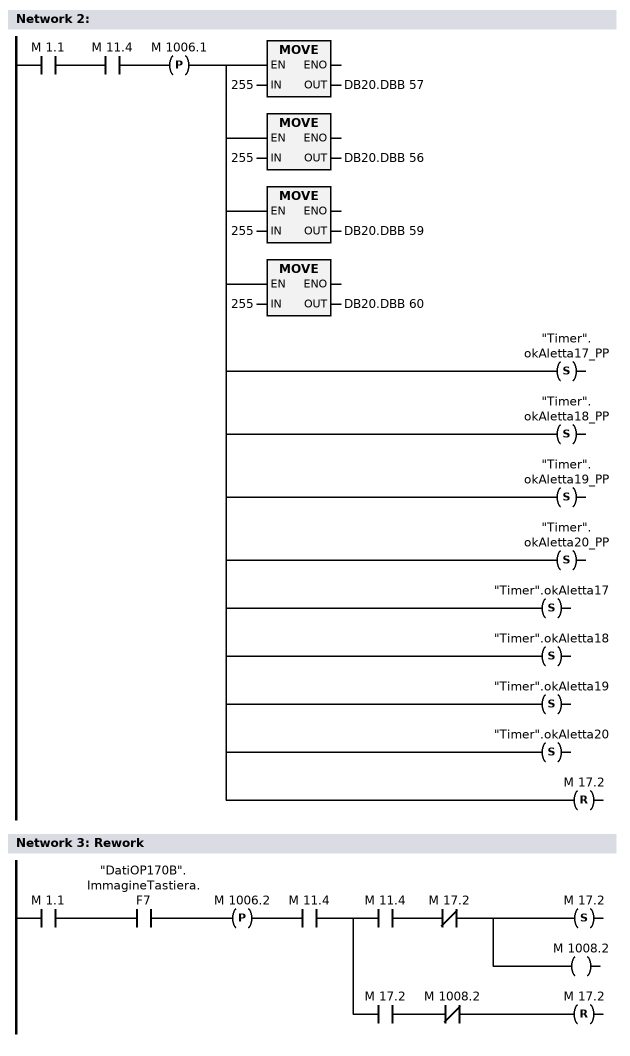
NETWORK
TITLE =
      A     M 1.1;
      A     M 11.4;
      FP    M 1006.1;
      =     L 0.0;
      A     L 0.0;
      JNB   _001;
      L     255;
      T     DB20.DBB 57;
_001: NOP   0;
      A     L 0.0;
      JNB   _002;
      L     255;
      T     DB20.DBB 56;
_002: NOP   0;
      A     L 0.0;
      JNB   _003;
      L     255;
      T     DB20.DBB 59;
_003: NOP   0;
      A     L 0.0;
      JNB   _004;
      L     255;
      T     DB20.DBB 60;
_004: NOP   0;
      A     L 0.0;
      BLD   102;
      S     "Timer".okAletta17_PP;
      A     L 0.0;
      BLD   102;
      S     "Timer".okAletta18_PP;
      A     L 0.0;
      BLD   102;
      S     "Timer".okAletta19_PP;
      A     L 0.0;
      BLD   102;
      S     "Timer".okAletta20_PP;
      A     L 0.0;
      BLD   102;
      S     "Timer".okAletta17;
      A     L 0.0;
      BLD   102;
      S     "Timer".okAletta18;
      A     L 0.0;
      BLD   102;
      S     "Timer".okAletta19;
      A     L 0.0;
      BLD   102;
      S     "Timer".okAletta20;
      A     L 0.0;
      BLD   102;
      R     M 17.2;
NETWORK
TITLE = Rework
      A     M 1.1;
      A     "DatiOP170B".ImmagineTastiera.F7;
      FP    M 1006.2;
      A     M 11.4;
      =     L 0.0;
      A     L 0.0;
      A     M 11.4;
      AN    M 17.2;
      S     M 17.2;
      =     M 1008.2;
      A     L 0.0;
      A     M 17.2;
      AN    M 1008.2;
      R     M 17.2;
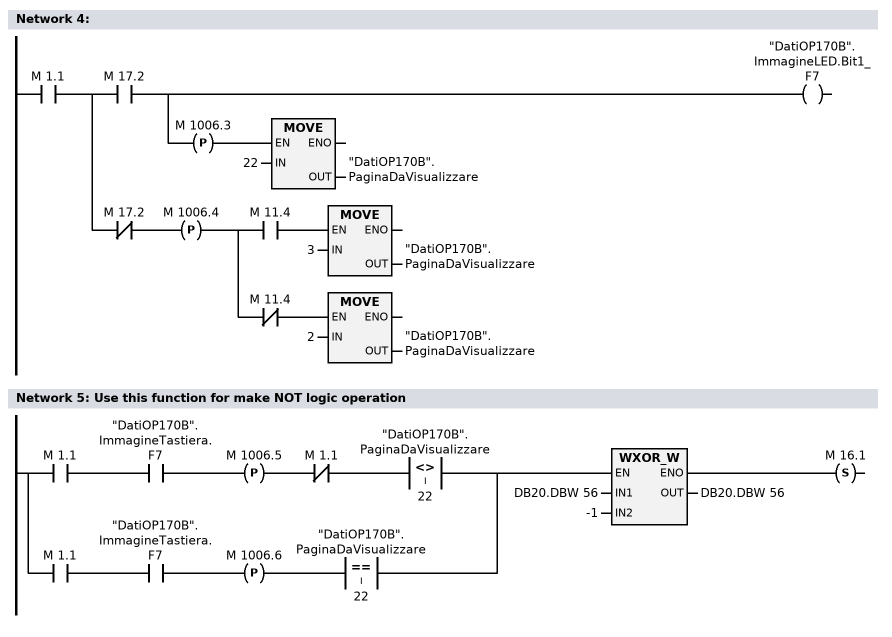
NETWORK
TITLE =
      A     M 1.1;
      =     L 0.0;
      A     L 0.0;
      A     M 17.2;
      =     L 0.1;
      A     L 0.1;
      BLD   102;
      =     "DatiOP170B".ImmagineLED.Bit1_F7;
      A     L 0.1;
      FP    M 1006.3;
      JNB   _005;
      L     22;
      T     "DatiOP170B".PaginaDaVisualizzare;
_005: NOP   0;
      A     L 0.0;
      AN    M 17.2;
      FP    M 1006.4;
      =     L 0.1;
      A     L 0.1;
      A     M 11.4;
      JNB   _006;
      L     3;
      T     "DatiOP170B".PaginaDaVisualizzare;
_006: NOP   0;
      A     L 0.1;
      AN    M 11.4;
      JNB   _007;
      L     2;
      T     "DatiOP170B".PaginaDaVisualizzare;
_007: NOP   0;
NETWORK
TITLE = Use this function for make NOT logic operation
//for invert functionality for operator
      A(;
      A     M 1.1;
      A     "DatiOP170B".ImmagineTastiera.F7;
      FP    M 1006.5;
      AN    M 1.1;
      A(;
      L     "DatiOP170B".PaginaDaVisualizzare;
      L     22;
      <>I;
      );
      O(;
      A     M 1.1;
      A     "DatiOP170B".ImmagineTastiera.F7;
      FP    M 1006.6;
      A(;
      L     "DatiOP170B".PaginaDaVisualizzare;
      L     22;
      ==I;
      );
      );
      );
      JNB   _008;
      L     DB20.DBW 56;
      L     -1;
      XOW;
      T     DB20.DBW 56;
      SET;
      SAVE;
      CLR;
_008: A     BR;
      S     M 16.1;
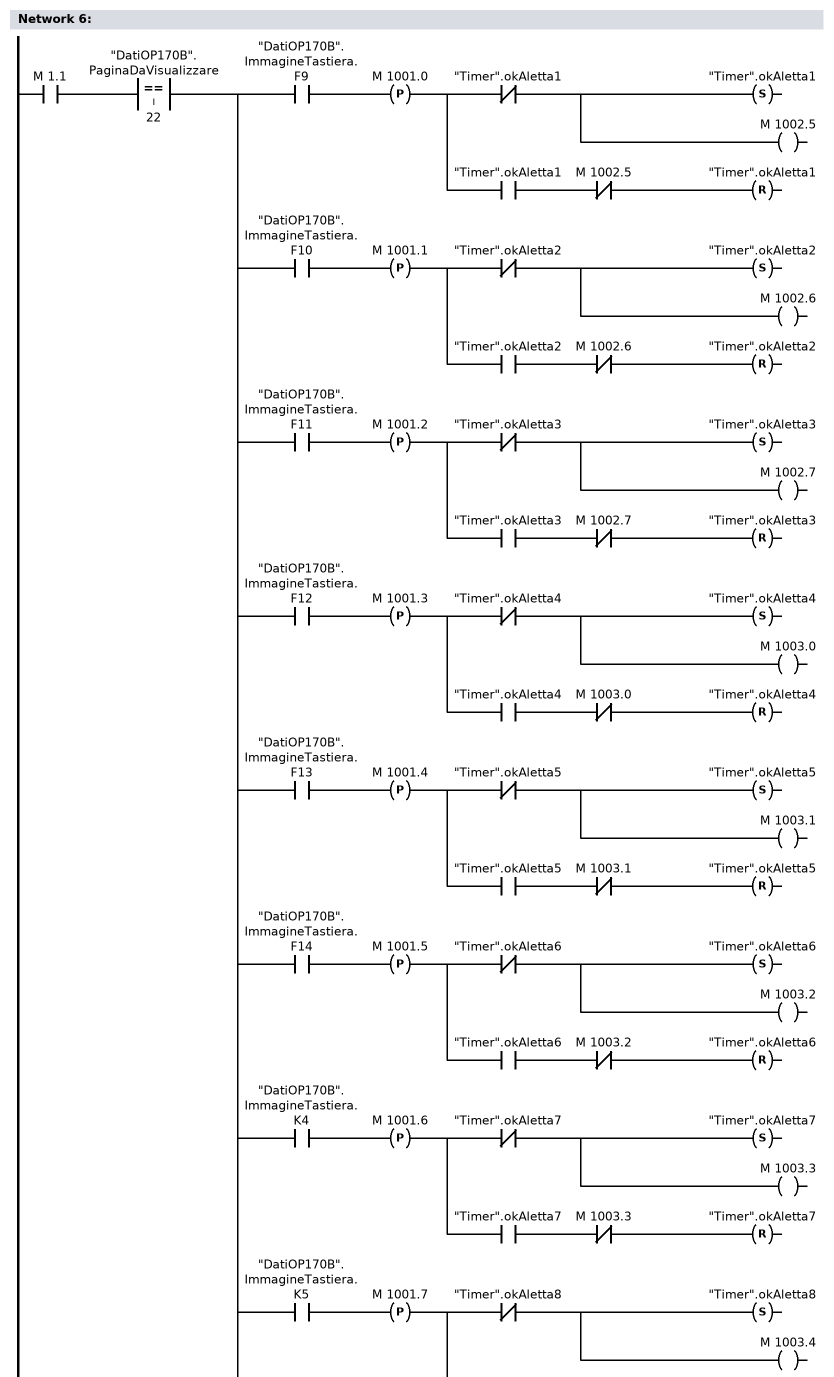
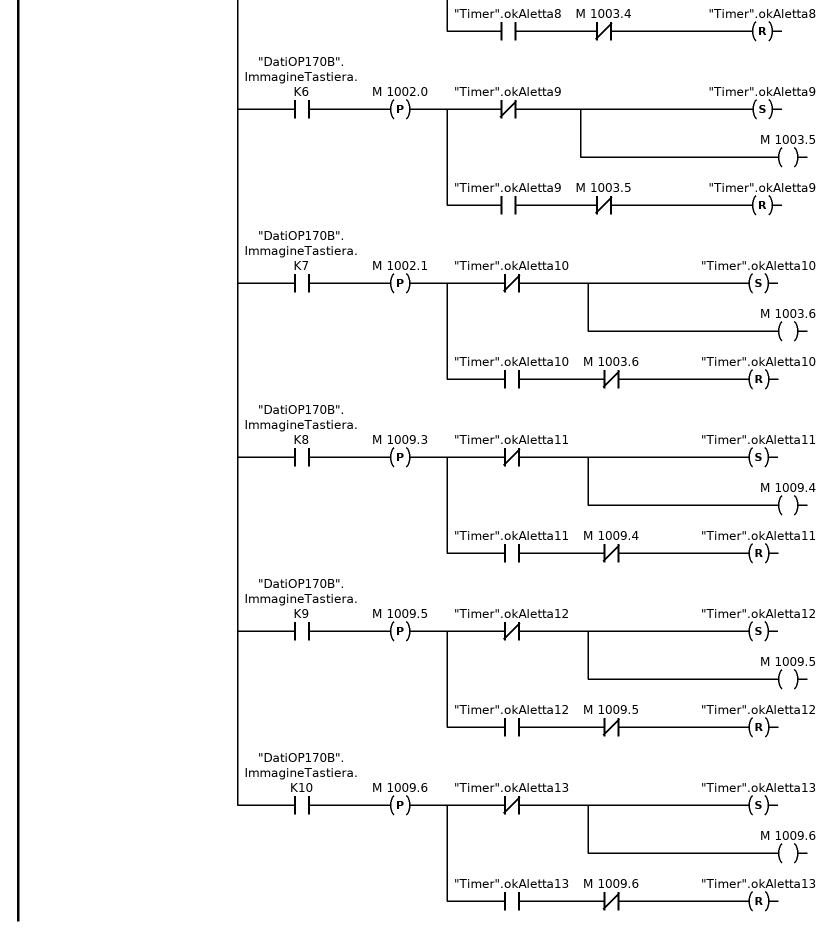
NETWORK
TITLE =
      A     M 1.1;
      A(;
      L     "DatiOP170B".PaginaDaVisualizzare;
      L     22;
      ==I;
      );
      =     L 0.0;
      A     L 0.0;
      A     "DatiOP170B".ImmagineTastiera.F9;
      FP    M 1001.0;
      =     L 0.1;
      A     L 0.1;
      AN    "Timer".okAletta1;
      S     "Timer".okAletta1;
      =     M 1002.5;
      A     L 0.1;
      A     "Timer".okAletta1;
      AN    M 1002.5;
      R     "Timer".okAletta1;
      A     L 0.0;
      A     "DatiOP170B".ImmagineTastiera.F10;
      FP    M 1001.1;
      =     L 0.1;
      A     L 0.1;
      AN    "Timer".okAletta2;
      S     "Timer".okAletta2;
      =     M 1002.6;
      A     L 0.1;
      A     "Timer".okAletta2;
      AN    M 1002.6;
      R     "Timer".okAletta2;
      A     L 0.0;
      A     "DatiOP170B".ImmagineTastiera.F11;
      FP    M 1001.2;
      =     L 0.1;
      A     L 0.1;
      AN    "Timer".okAletta3;
      S     "Timer".okAletta3;
      =     M 1002.7;
      A     L 0.1;
      A     "Timer".okAletta3;
      AN    M 1002.7;
      R     "Timer".okAletta3;
      A     L 0.0;
      A     "DatiOP170B".ImmagineTastiera.F12;
      FP    M 1001.3;
      =     L 0.1;
      A     L 0.1;
      AN    "Timer".okAletta4;
      S     "Timer".okAletta4;
      =     M 1003.0;
      A     L 0.1;
      A     "Timer".okAletta4;
      AN    M 1003.0;
      R     "Timer".okAletta4;
      A     L 0.0;
      A     "DatiOP170B".ImmagineTastiera.F13;
      FP    M 1001.4;
      =     L 0.1;
      A     L 0.1;
      AN    "Timer".okAletta5;
      S     "Timer".okAletta5;
      =     M 1003.1;
      A     L 0.1;
      A     "Timer".okAletta5;
      AN    M 1003.1;
      R     "Timer".okAletta5;
      A     L 0.0;
      A     "DatiOP170B".ImmagineTastiera.F14;
      FP    M 1001.5;
      =     L 0.1;
      A     L 0.1;
      AN    "Timer".okAletta6;
      S     "Timer".okAletta6;
      =     M 1003.2;
      A     L 0.1;
      A     "Timer".okAletta6;
      AN    M 1003.2;
      R     "Timer".okAletta6;
      A     L 0.0;
      A     "DatiOP170B".ImmagineTastiera.K4;
      FP    M 1001.6;
      =     L 0.1;
      A     L 0.1;
      AN    "Timer".okAletta7;
      S     "Timer".okAletta7;
      =     M 1003.3;
      A     L 0.1;
      A     "Timer".okAletta7;
      AN    M 1003.3;
      R     "Timer".okAletta7;
      A     L 0.0;
      A     "DatiOP170B".ImmagineTastiera.K5;
      FP    M 1001.7;
      =     L 0.1;
      A     L 0.1;
      AN    "Timer".okAletta8;
      S     "Timer".okAletta8;
      =     M 1003.4;
      A     L 0.1;
      A     "Timer".okAletta8;
      AN    M 1003.4;
      R     "Timer".okAletta8;
      A     L 0.0;
      A     "DatiOP170B".ImmagineTastiera.K6;
      FP    M 1002.0;
      =     L 0.1;
      A     L 0.1;
      AN    "Timer".okAletta9;
      S     "Timer".okAletta9;
      =     M 1003.5;
      A     L 0.1;
      A     "Timer".okAletta9;
      AN    M 1003.5;
      R     "Timer".okAletta9;
      A     L 0.0;
      A     "DatiOP170B".ImmagineTastiera.K7;
      FP    M 1002.1;
      =     L 0.1;
      A     L 0.1;
      AN    "Timer".okAletta10;
      S     "Timer".okAletta10;
      =     M 1003.6;
      A     L 0.1;
      A     "Timer".okAletta10;
      AN    M 1003.6;
      R     "Timer".okAletta10;
      A     L 0.0;
      A     "DatiOP170B".ImmagineTastiera.K8;
      FP    M 1009.3;
      =     L 0.1;
      A     L 0.1;
      AN    "Timer".okAletta11;
      S     "Timer".okAletta11;
      =     M 1009.4;
      A     L 0.1;
      A     "Timer".okAletta11;
      AN    M 1009.4;
      R     "Timer".okAletta11;
      A     L 0.0;
      A     "DatiOP170B".ImmagineTastiera.K9;
      FP    M 1009.5;
      =     L 0.1;
      A     L 0.1;
      AN    "Timer".okAletta12;
      S     "Timer".okAletta12;
      =     M 1009.5;
      A     L 0.1;
      A     "Timer".okAletta12;
      AN    M 1009.5;
      R     "Timer".okAletta12;
      A     L 0.0;
      A     "DatiOP170B".ImmagineTastiera.K10;
      FP    M 1009.6;
      =     L 0.1;
      A     L 0.1;
      AN    "Timer".okAletta13;
      S     "Timer".okAletta13;
      =     M 1009.6;
      A     L 0.1;
      A     "Timer".okAletta13;
      AN    M 1009.6;
      R     "Timer".okAletta13;
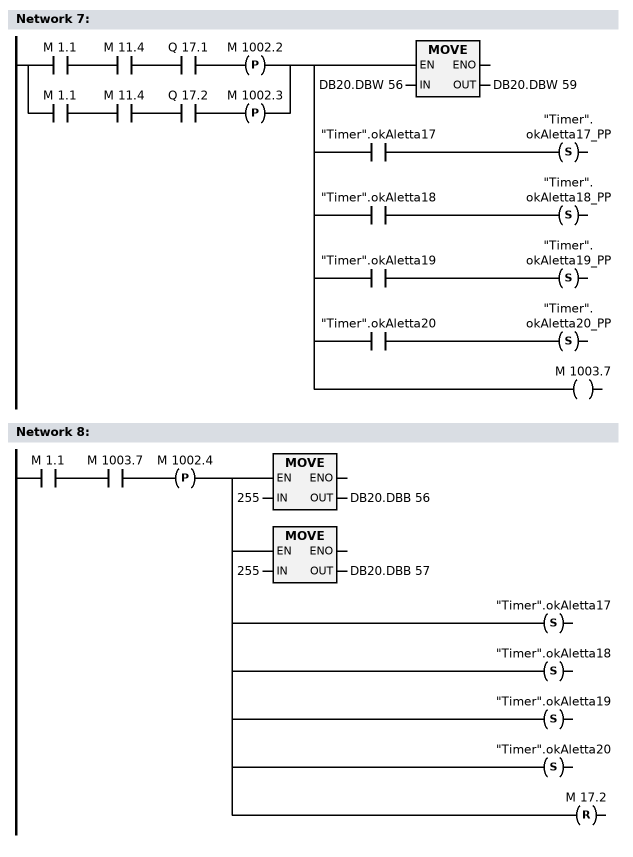
NETWORK
TITLE =
      A     M 1.1;
      A     M 11.4;
      A     Q 17.1;
      FP    M 1002.2;
      O(;
      A     M 1.1;
      A     M 11.4;
      A     Q 17.2;
      FP    M 1002.3;
      );
      =     L 0.0;
      A     L 0.0;
      JNB   _009;
      L     DB20.DBW 56;
      T     DB20.DBW 59;
_009: NOP   0;
      A     L 0.0;
      A     "Timer".okAletta17;
      S     "Timer".okAletta17_PP;
      A     L 0.0;
      A     "Timer".okAletta18;
      S     "Timer".okAletta18_PP;
      A     L 0.0;
      A     "Timer".okAletta19;
      S     "Timer".okAletta19_PP;
      A     L 0.0;
      A     "Timer".okAletta20;
      S     "Timer".okAletta20_PP;
      A     L 0.0;
      BLD   102;
      =     M 1003.7;
NETWORK
TITLE =
      A     M 1.1;
      A     M 1003.7;
      FP    M 1002.4;
      =     L 0.0;
      A     L 0.0;
      JNB   _00a;
      L     255;
      T     DB20.DBB 56;
_00a: NOP   0;
      A     L 0.0;
      JNB   _00b;
      L     255;
      T     DB20.DBB 57;
_00b: NOP   0;
      A     L 0.0;
      BLD   102;
      S     "Timer".okAletta17;
      A     L 0.0;
      BLD   102;
      S     "Timer".okAletta18;
      A     L 0.0;
      BLD   102;
      S     "Timer".okAletta19;
      A     L 0.0;
      BLD   102;
      S     "Timer".okAletta20;
      A     L 0.0;
      BLD   102;
      R     M 17.2;
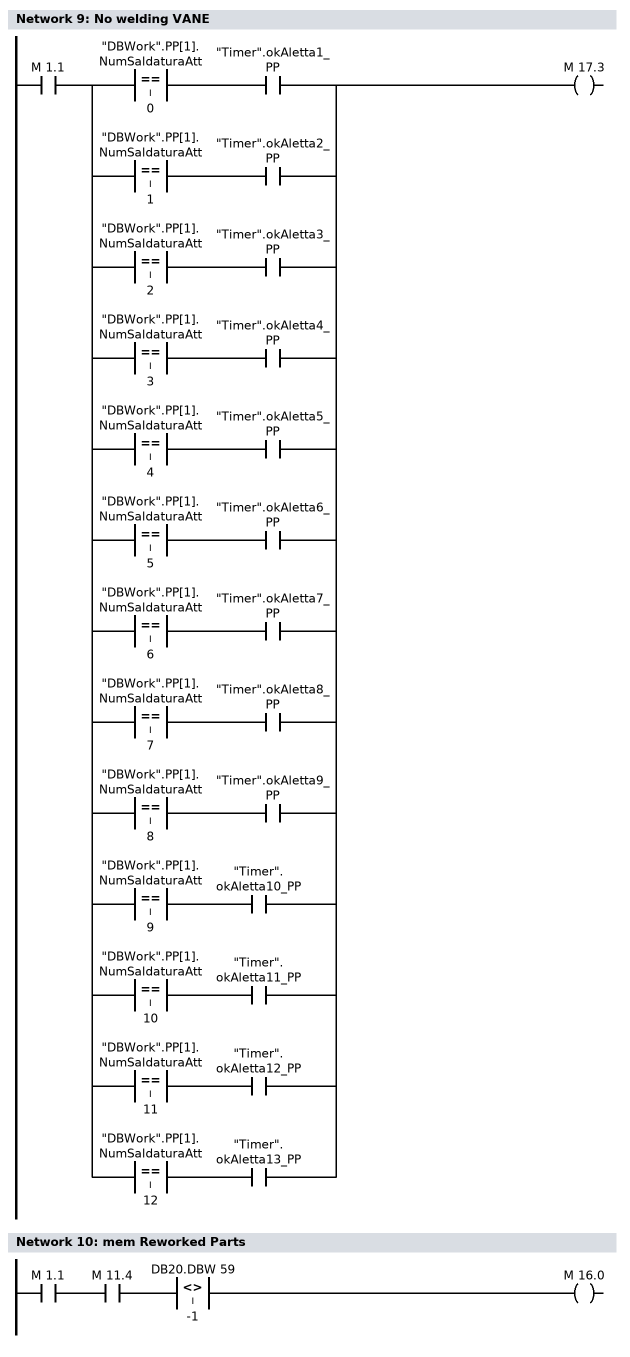
NETWORK
TITLE = No welding VANE
      A     M 1.1;
      A(;
      A(;
      L     "DBWork".PP[1].NumSaldaturaAtt;
      L     0;
      ==I;
      );
      A     "Timer".okAletta1_PP;
      O;
      A(;
      L     "DBWork".PP[1].NumSaldaturaAtt;
      L     1;
      ==I;
      );
      A     "Timer".okAletta2_PP;
      O;
      A(;
      L     "DBWork".PP[1].NumSaldaturaAtt;
      L     2;
      ==I;
      );
      A     "Timer".okAletta3_PP;
      O;
      A(;
      L     "DBWork".PP[1].NumSaldaturaAtt;
      L     3;
      ==I;
      );
      A     "Timer".okAletta4_PP;
      O;
      A(;
      L     "DBWork".PP[1].NumSaldaturaAtt;
      L     4;
      ==I;
      );
      A     "Timer".okAletta5_PP;
      O;
      A(;
      L     "DBWork".PP[1].NumSaldaturaAtt;
      L     5;
      ==I;
      );
      A     "Timer".okAletta6_PP;
      O;
      A(;
      L     "DBWork".PP[1].NumSaldaturaAtt;
      L     6;
      ==I;
      );
      A     "Timer".okAletta7_PP;
      O;
      A(;
      L     "DBWork".PP[1].NumSaldaturaAtt;
      L     7;
      ==I;
      );
      A     "Timer".okAletta8_PP;
      O;
      A(;
      L     "DBWork".PP[1].NumSaldaturaAtt;
      L     8;
      ==I;
      );
      A     "Timer".okAletta9_PP;
      O;
      A(;
      L     "DBWork".PP[1].NumSaldaturaAtt;
      L     9;
      ==I;
      );
      A     "Timer".okAletta10_PP;
      O;
      A(;
      L     "DBWork".PP[1].NumSaldaturaAtt;
      L     10;
      ==I;
      );
      A     "Timer".okAletta11_PP;
      O;
      A(;
      L     "DBWork".PP[1].NumSaldaturaAtt;
      L     11;
      ==I;
      );
      A     "Timer".okAletta12_PP;
      O;
      A(;
      L     "DBWork".PP[1].NumSaldaturaAtt;
      L     12;
      ==I;
      );
      A     "Timer".okAletta13_PP;
      );
      =     M 17.3;
NETWORK
TITLE = mem Reworked Parts
      A     M 1.1;
      A     M 11.4;
      A(;
      L     DB20.DBW 59;
      L     -1;
      <>I;
      );
      =     M 16.0;
END_FUNCTION

FUNCTION "FC81 - GEST AXIS" : VOID	// FC 81
VERSION : 0.1
VAR_TEMP
  AttualPos : DINT ;
  AttualPosR : REAL ;
  Override : INT ;
  AuxRelative : DINT ;
  JogRelative : BOOL ;
END_VAR
BEGIN
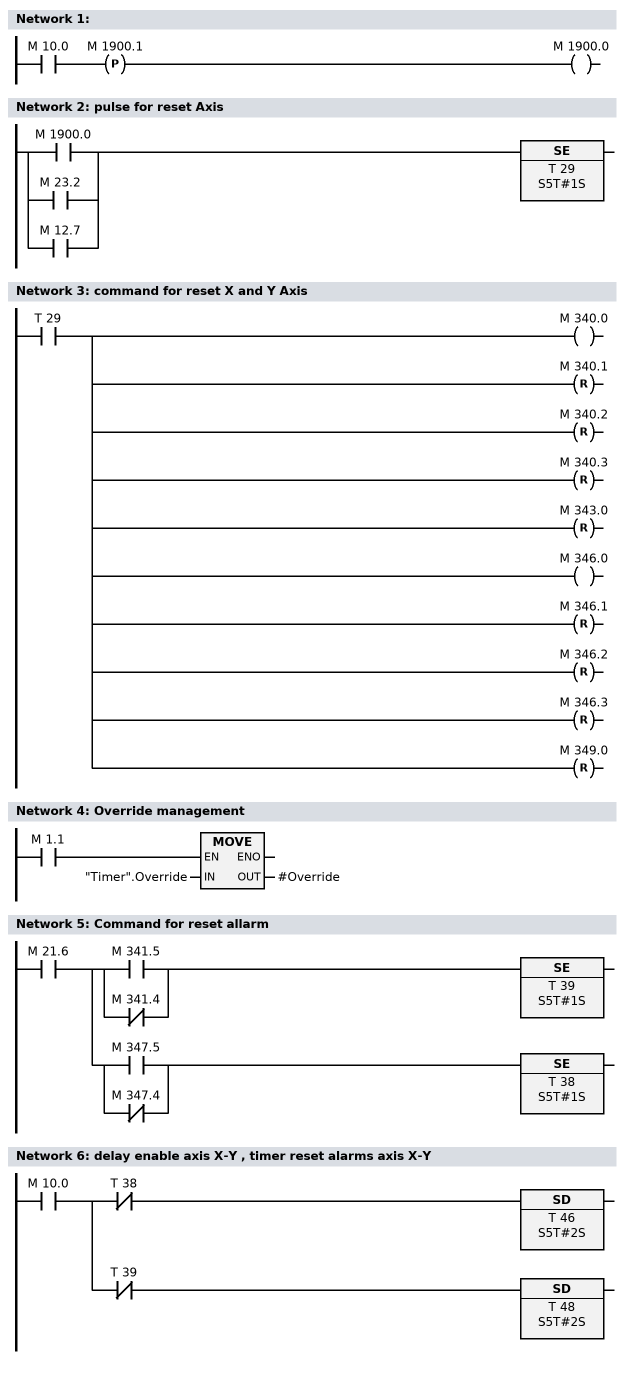
NETWORK
TITLE =
      A     M 10.0;
      FP    M 1900.1;
      =     M 1900.0;
NETWORK
TITLE = pulse for reset Axis
      O     M 1900.0;
      O     M 23.2;
      O     M 12.7;
      L     S5T#1S;
      SE    T 29;
NETWORK
TITLE = command for reset X and Y Axis
      A     T 29;
      =     M 340.0;
      R     M 340.1;
      R     M 340.2;
      R     M 340.3;
      R     M 343.0;
      =     M 346.0;
      R     M 346.1;
      R     M 346.2;
      R     M 346.3;
      R     M 349.0;
NETWORK
TITLE = Override management
//"DatiMacchina".AcesXYZC_Override_Aux
      A     M 1.1;
      JNB   _001;
      L     "Timer".Override;
      T     #Override;
_001: NOP   0;
NETWORK
TITLE = Command for reset allarm
      A     M 21.6;
      =     L 15.0;
      A     L 15.0;
      A(;
      O     M 341.5;
      ON    M 341.4;
      );
      L     S5T#1S;
      SE    T 39;
      A     L 15.0;
      A(;
      O     M 347.5;
      ON    M 347.4;
      );
      L     S5T#1S;
      SE    T 38;
NETWORK
TITLE = delay enable axis X-Y , timer reset alarms axis X-Y
      A     M 10.0;
      =     L 15.0;
      A     L 15.0;
      AN    T 38;
      L     S5T#2S;
      SD    T 46;
      A     L 15.0;
      AN    T 39;
      L     S5T#2S;
      SD    T 48;
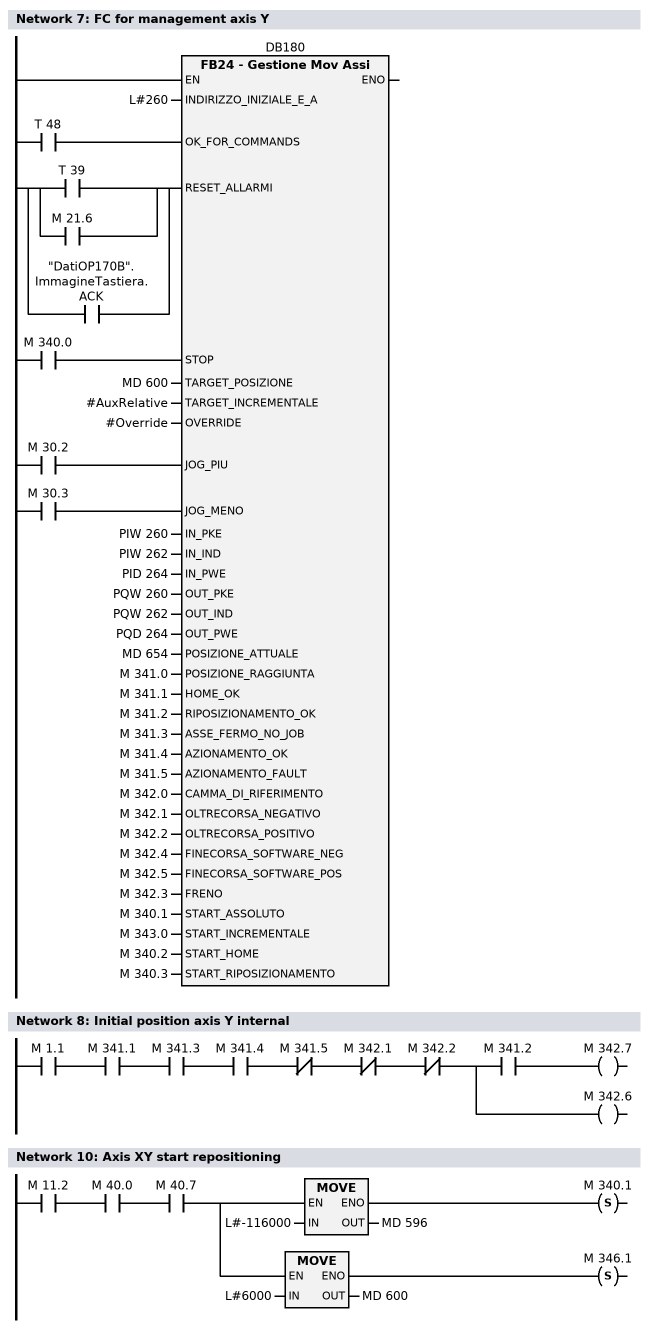
NETWORK
TITLE = FC for management axis Y
      A     T 48;
      =     L 15.0;
      BLD   103;
      A(;
      O     T 39;
      O     M 21.6;
      O     "DatiOP170B".ImmagineTastiera.ACK;
      );
      =     L 15.1;
      BLD   103;
      A     M 340.0;
      =     L 15.2;
      BLD   103;
      A     M 30.2;
      =     L 15.3;
      BLD   103;
      A     M 30.3;
      =     L 15.4;
      BLD   103;
      CALL  "FB24 - Gestione Mov Assi" , "DB180" (
           INDIRIZZO_INIZIALE_E_A   := L#260,
           OK_FOR_COMMANDS          := L 15.0,
           RESET_ALLARMI            := L 15.1,
           STOP                     := L 15.2,
           TARGET_POSIZIONE         := MD 600,
           TARGET_INCREMENTALE      := #AuxRelative,
           OVERRIDE                 := #Override,
           JOG_PIU                  := L 15.3,
           JOG_MENO                 := L 15.4,
           IN_PKE                   := PIW 260,
           IN_IND                   := PIW 262,
           IN_PWE                   := PID 264,
           OUT_PKE                  := PQW 260,
           OUT_IND                  := PQW 262,
           OUT_PWE                  := PQD 264,
           POSIZIONE_ATTUALE        := MD 654,
           POSIZIONE_RAGGIUNTA      := M 341.0,
           HOME_OK                  := M 341.1,
           RIPOSIZIONAMENTO_OK      := M 341.2,
           ASSE_FERMO_NO_JOB        := M 341.3,
           AZIONAMENTO_OK           := M 341.4,
           AZIONAMENTO_FAULT        := M 341.5,
           CAMMA_DI_RIFERIMENTO     := M 342.0,
           OLTRECORSA_NEGATIVO      := M 342.1,
           OLTRECORSA_POSITIVO      := M 342.2,
           FINECORSA_SOFTWARE_NEG   := M 342.4,
           FINECORSA_SOFTWARE_POS   := M 342.5,
           FRENO                    := M 342.3,
           START_ASSOLUTO           := M 340.1,
           START_INCREMENTALE       := M 343.0,
           START_HOME               := M 340.2,
           START_RIPOSIZIONAMENTO   := M 340.3);
      NOP   0;
NETWORK
TITLE = Initial position axis Y internal
      A     M 1.1;
      A     M 341.1;
      A     M 341.3;
      A     M 341.4;
      AN    M 341.5;
      AN    M 342.1;
      AN    M 342.2;
      =     L 15.0;
      A     L 15.0;
      A     M 341.2;
      =     M 342.7;
      A     L 15.0;
      BLD   102;
      =     M 342.6;
NETWORK
TITLE = Axis X Management
NETWORK
TITLE = Axis XY start repositioning
      A     M 11.2;
      A     M 40.0;
      A     M 40.7;
      =     L 15.0;
      A     L 15.0;
      JNB   _002;
      L     L#-116000;
      T     MD 596;
      SET;
      SAVE;
      CLR;
_002: A     BR;
      S     M 340.1;
      A     L 15.0;
      JNB   _003;
      L     L#6000;
      T     MD 600;
      SET;
      SAVE;
      CLR;
_003: A     BR;
      S     M 346.1;
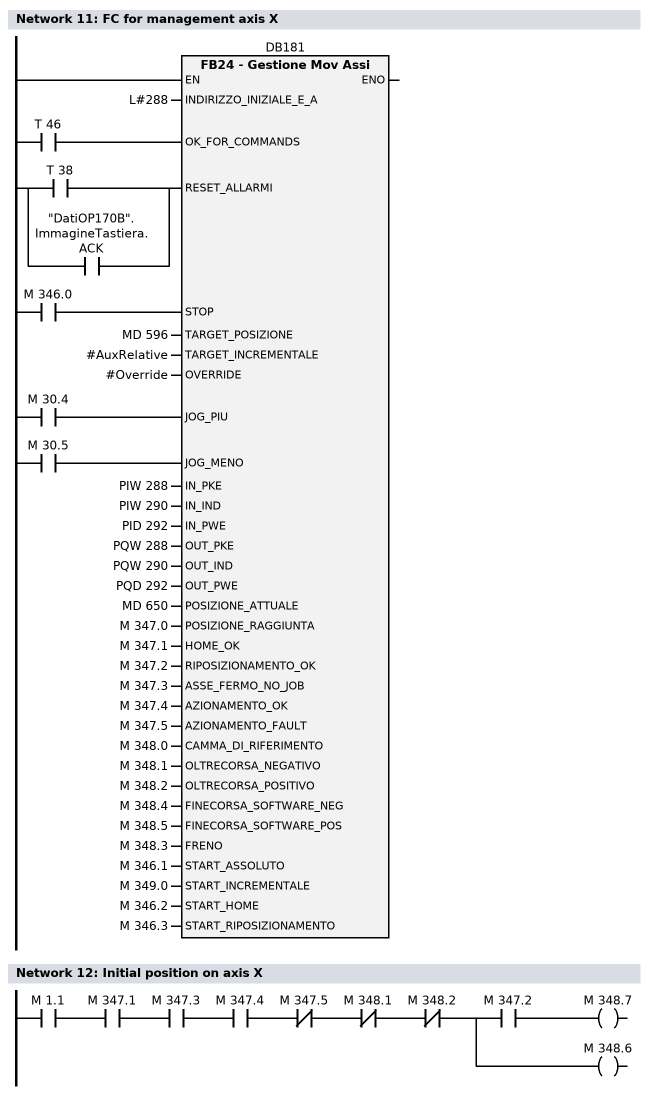
NETWORK
TITLE = FC for management axis X
      A     T 46;
      =     L 15.0;
      BLD   103;
      A(;
      O     T 38;
      O     "DatiOP170B".ImmagineTastiera.ACK;
      );
      =     L 15.1;
      BLD   103;
      A     M 346.0;
      =     L 15.2;
      BLD   103;
      A     M 30.4;
      =     L 15.3;
      BLD   103;
      A     M 30.5;
      =     L 15.4;
      BLD   103;
      CALL  "FB24 - Gestione Mov Assi" , "DB181" (
           INDIRIZZO_INIZIALE_E_A   := L#288,
           OK_FOR_COMMANDS          := L 15.0,
           RESET_ALLARMI            := L 15.1,
           STOP                     := L 15.2,
           TARGET_POSIZIONE         := MD 596,
           TARGET_INCREMENTALE      := #AuxRelative,
           OVERRIDE                 := #Override,
           JOG_PIU                  := L 15.3,
           JOG_MENO                 := L 15.4,
           IN_PKE                   := PIW 288,
           IN_IND                   := PIW 290,
           IN_PWE                   := PID 292,
           OUT_PKE                  := PQW 288,
           OUT_IND                  := PQW 290,
           OUT_PWE                  := PQD 292,
           POSIZIONE_ATTUALE        := MD 650,
           POSIZIONE_RAGGIUNTA      := M 347.0,
           HOME_OK                  := M 347.1,
           RIPOSIZIONAMENTO_OK      := M 347.2,
           ASSE_FERMO_NO_JOB        := M 347.3,
           AZIONAMENTO_OK           := M 347.4,
           AZIONAMENTO_FAULT        := M 347.5,
           CAMMA_DI_RIFERIMENTO     := M 348.0,
           OLTRECORSA_NEGATIVO      := M 348.1,
           OLTRECORSA_POSITIVO      := M 348.2,
           FINECORSA_SOFTWARE_NEG   := M 348.4,
           FINECORSA_SOFTWARE_POS   := M 348.5,
           FRENO                    := M 348.3,
           START_ASSOLUTO           := M 346.1,
           START_INCREMENTALE       := M 349.0,
           START_HOME               := M 346.2,
           START_RIPOSIZIONAMENTO   := M 346.3);
      NOP   0;
NETWORK
TITLE = Initial position on axis X
      A     M 1.1;
      A     M 347.1;
      A     M 347.3;
      A     M 347.4;
      AN    M 347.5;
      AN    M 348.1;
      AN    M 348.2;
      =     L 15.0;
      A     L 15.0;
      A     M 347.2;
      =     M 348.7;
      A     L 15.0;
      BLD   102;
      =     M 348.6;
END_FUNCTION

FUNCTION "FC117 - ERROR TOOL" : VOID	// FC 117
VERSION : 0.1
BEGIN
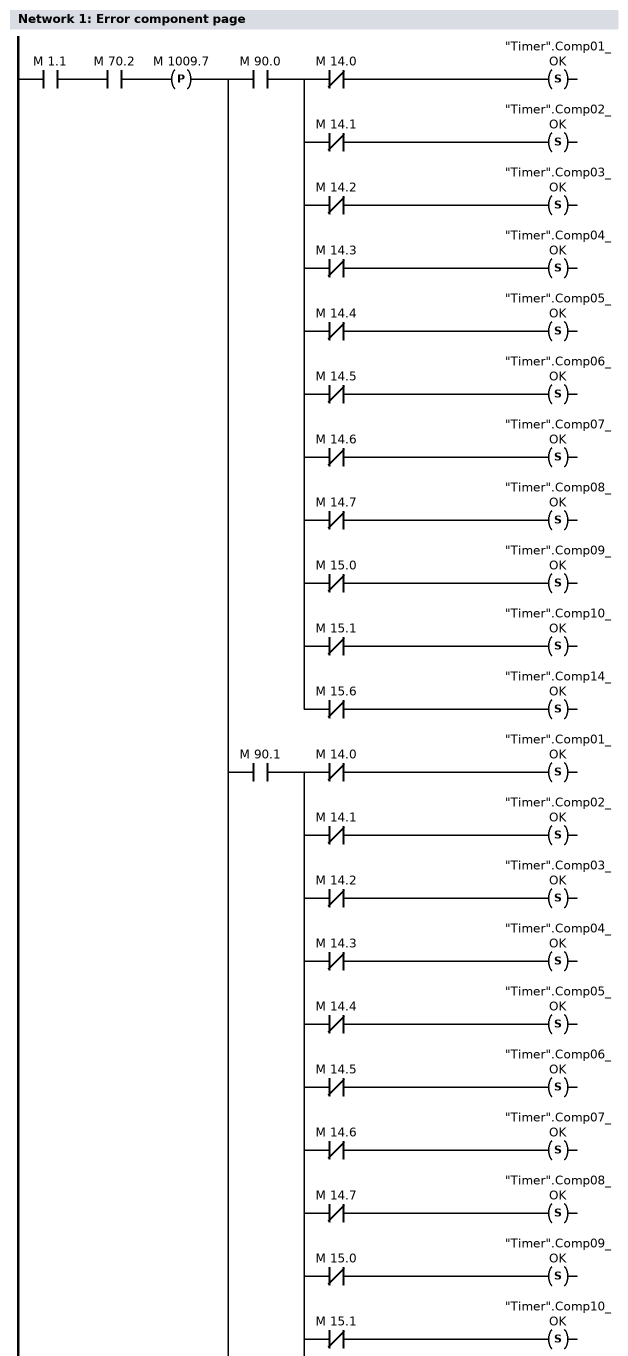
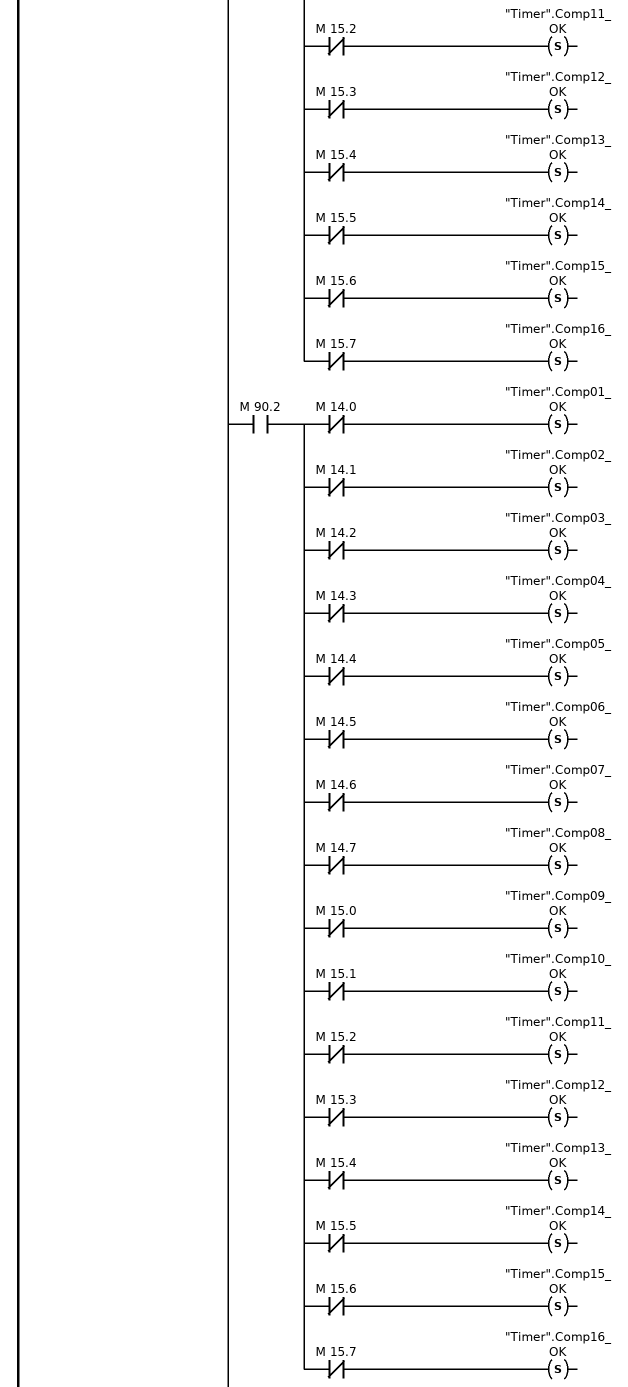
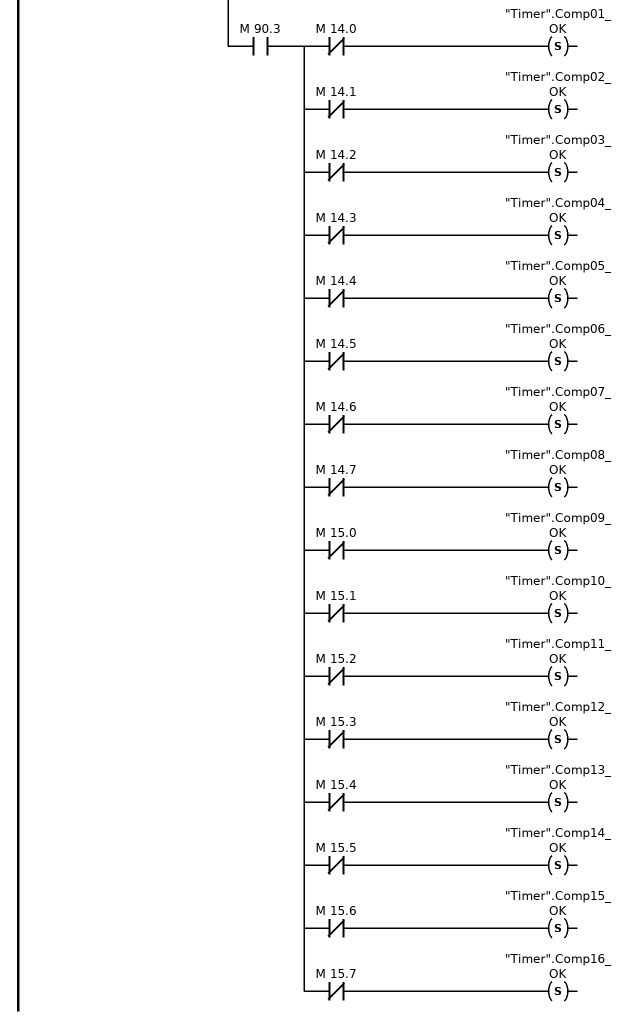
NETWORK
TITLE = Error component page
      A     M 1.1;
      A     M 70.2;
      FP    M 1009.7;
      =     L 0.0;
      A     L 0.0;
      A     M 90.0;
      =     L 0.1;
      A     L 0.1;
      AN    M 14.0;
      S     "Timer".Comp01_OK;
      A     L 0.1;
      AN    M 14.1;
      S     "Timer".Comp02_OK;
      A     L 0.1;
      AN    M 14.2;
      S     "Timer".Comp03_OK;
      A     L 0.1;
      AN    M 14.3;
      S     "Timer".Comp04_OK;
      A     L 0.1;
      AN    M 14.4;
      S     "Timer".Comp05_OK;
      A     L 0.1;
      AN    M 14.5;
      S     "Timer".Comp06_OK;
      A     L 0.1;
      AN    M 14.6;
      S     "Timer".Comp07_OK;
      A     L 0.1;
      AN    M 14.7;
      S     "Timer".Comp08_OK;
      A     L 0.1;
      AN    M 15.0;
      S     "Timer".Comp09_OK;
      A     L 0.1;
      AN    M 15.1;
      S     "Timer".Comp10_OK;
      A     L 0.1;
      AN    M 15.6;
      S     "Timer".Comp14_OK;
      A     L 0.0;
      A     M 90.1;
      =     L 0.1;
      A     L 0.1;
      AN    M 14.0;
      S     "Timer".Comp01_OK;
      A     L 0.1;
      AN    M 14.1;
      S     "Timer".Comp02_OK;
      A     L 0.1;
      AN    M 14.2;
      S     "Timer".Comp03_OK;
      A     L 0.1;
      AN    M 14.3;
      S     "Timer".Comp04_OK;
      A     L 0.1;
      AN    M 14.4;
      S     "Timer".Comp05_OK;
      A     L 0.1;
      AN    M 14.5;
      S     "Timer".Comp06_OK;
      A     L 0.1;
      AN    M 14.6;
      S     "Timer".Comp07_OK;
      A     L 0.1;
      AN    M 14.7;
      S     "Timer".Comp08_OK;
      A     L 0.1;
      AN    M 15.0;
      S     "Timer".Comp09_OK;
      A     L 0.1;
      AN    M 15.1;
      S     "Timer".Comp10_OK;
      A     L 0.1;
      AN    M 15.2;
      S     "Timer".Comp11_OK;
      A     L 0.1;
      AN    M 15.3;
      S     "Timer".Comp12_OK;
      A     L 0.1;
      AN    M 15.4;
      S     "Timer".Comp13_OK;
      A     L 0.1;
      AN    M 15.5;
      S     "Timer".Comp14_OK;
      A     L 0.1;
      AN    M 15.6;
      S     "Timer".Comp15_OK;
      A     L 0.1;
      AN    M 15.7;
      S     "Timer".Comp16_OK;
      A     L 0.0;
      A     M 90.2;
      =     L 0.1;
      A     L 0.1;
      AN    M 14.0;
      S     "Timer".Comp01_OK;
      A     L 0.1;
      AN    M 14.1;
      S     "Timer".Comp02_OK;
      A     L 0.1;
      AN    M 14.2;
      S     "Timer".Comp03_OK;
      A     L 0.1;
      AN    M 14.3;
      S     "Timer".Comp04_OK;
      A     L 0.1;
      AN    M 14.4;
      S     "Timer".Comp05_OK;
      A     L 0.1;
      AN    M 14.5;
      S     "Timer".Comp06_OK;
      A     L 0.1;
      AN    M 14.6;
      S     "Timer".Comp07_OK;
      A     L 0.1;
      AN    M 14.7;
      S     "Timer".Comp08_OK;
      A     L 0.1;
      AN    M 15.0;
      S     "Timer".Comp09_OK;
      A     L 0.1;
      AN    M 15.1;
      S     "Timer".Comp10_OK;
      A     L 0.1;
      AN    M 15.2;
      S     "Timer".Comp11_OK;
      A     L 0.1;
      AN    M 15.3;
      S     "Timer".Comp12_OK;
      A     L 0.1;
      AN    M 15.4;
      S     "Timer".Comp13_OK;
      A     L 0.1;
      AN    M 15.5;
      S     "Timer".Comp14_OK;
      A     L 0.1;
      AN    M 15.6;
      S     "Timer".Comp15_OK;
      A     L 0.1;
      AN    M 15.7;
      S     "Timer".Comp16_OK;
      A     L 0.0;
      A     M 90.3;
      =     L 0.1;
      A     L 0.1;
      AN    M 14.0;
      S     "Timer".Comp01_OK;
      A     L 0.1;
      AN    M 14.1;
      S     "Timer".Comp02_OK;
      A     L 0.1;
      AN    M 14.2;
      S     "Timer".Comp03_OK;
      A     L 0.1;
      AN    M 14.3;
      S     "Timer".Comp04_OK;
      A     L 0.1;
      AN    M 14.4;
      S     "Timer".Comp05_OK;
      A     L 0.1;
      AN    M 14.5;
      S     "Timer".Comp06_OK;
      A     L 0.1;
      AN    M 14.6;
      S     "Timer".Comp07_OK;
      A     L 0.1;
      AN    M 14.7;
      S     "Timer".Comp08_OK;
      A     L 0.1;
      AN    M 15.0;
      S     "Timer".Comp09_OK;
      A     L 0.1;
      AN    M 15.1;
      S     "Timer".Comp10_OK;
      A     L 0.1;
      AN    M 15.2;
      S     "Timer".Comp11_OK;
      A     L 0.1;
      AN    M 15.3;
      S     "Timer".Comp12_OK;
      A     L 0.1;
      AN    M 15.4;
      S     "Timer".Comp13_OK;
      A     L 0.1;
      AN    M 15.5;
      S     "Timer".Comp14_OK;
      A     L 0.1;
      AN    M 15.6;
      S     "Timer".Comp15_OK;
      A     L 0.1;
      AN    M 15.7;
      S     "Timer".Comp16_OK;
END_FUNCTION

FUNCTION "TimeOut" : VOID	// FC 800
TITLE = Gestione timeout movimento
FAMILY : GCLib
NAME : TimeOut
VERSION : 1.0
VAR_INPUT
  Condizione1 : BOOL ;
  Condizione2 : BOOL ;
  Contatore : COUNTER ;
  Reset : BOOL ;
  Tempo_TimeOut : INT ;
END_VAR
VAR_IN_OUT
  TimeOut_Condizione1 : BOOL ;
  TimeOut_Condizione2 : BOOL ;
END_VAR
BEGIN
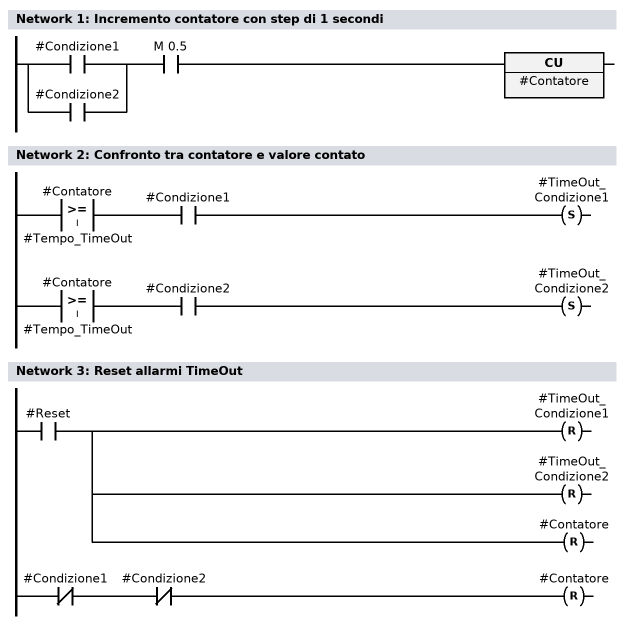
NETWORK
TITLE = Incremento contatore con step di 1 secondi
      A     #Condizione1;
      O     #Condizione2;
      A     M 0.5;
      CU    #Contatore;
NETWORK
TITLE = Confronto tra contatore e valore contato
      L     #Contatore;
      L     #Tempo_TimeOut;
      >=I;
      A     #Condizione1;
      S     #TimeOut_Condizione1;
      L     #Contatore;
      L     #Tempo_TimeOut;
      >=I;
      A     #Condizione2;
      S     #TimeOut_Condizione2;
NETWORK
TITLE = Reset allarmi TimeOut
      A     #Reset;
      R     #TimeOut_Condizione1;
      R     #TimeOut_Condizione2;
      R     #Contatore;
      AN    #Condizione1;
      AN    #Condizione2;
      R     #Contatore;
END_FUNCTION

DATA_BLOCK "DI_Balluff1"	// DB 5
VERSION : 0.0
"BALLUFF"
BEGIN
END_DATA_BLOCK

